// TIA Portal V17 export
// export: Created 2025-05-08T13:18:02.6118738Z, ExportSetting WithDefaults, DisplayName Totally Integrated Automation Portal, DisplayVersion V17 Update 8, DisplayName TIA Portal Openness, DisplayVersion V17 Update 8, DisplayName TIA Portal Version Control Interface, DisplayVersion V17, DisplayName SINAMICS Startdrive Advanced, DisplayVersion V17 SP2, DisplayName SINAMICS Startdrive G110M, G120, G120C, G120D, G120P, G115D, DisplayVersion V17 SP2, DisplayName SINAMICS Startdrive G130, G150, S120, S150, SINAMICS MV, S210, DisplayVersion V17 SP2, DisplayName STEP 7 Professional, DisplayVersion V17 Update 8, DisplayName SINUMERIK ONE STEP 7 Toolbox, DisplayVersion V17 Update 12, DisplayName SINUMERIK 840D sl STEP 7 Toolbox, DisplayVersion V17 Update 12, DisplayName STEP 7 Safety, DisplayVersion V17 Update 6, DisplayName WinCC Advanced, DisplayVersion V17 Update 8
FUNCTION "FC16016_METHOD_CALLS_U3_MEAS_STA_MEAS_R" : Void   // FC16016, LAD
{ S7_Optimized_Access := 'TRUE' }
VERSION : 0.1
// stored: AutoNumber false, IsIECCheckEnabled false, SetENOAutomatically false, UDAEnableTagReadback false
   VAR_TEMP
      AUX_WSTRING_PART_ID_MEAS_STA : WString;
      AUX_WCHARS : Array[0..63] of WChar;
      index : Int;
      AUX_ALARMS : Bool;
   END_VAR
   VAR CONSTANT
      VERSIONS_MAJOR : UInt := 2;
      VERSIONS_MINOR : UInt;
      FC_NUMBER : DInt := 16016;
   END_VAR
   VAR_TEMP   // added for the SCL form of the ladder/FBD networks
      _w1 : Bool;
      _w2 : Bool;
   END_VAR
BEGIN

REGION Network 1 (SCL): TRANSFORM TO WCHARS
   FOR #index := 0 TO 63 DO
       #AUX_WCHARS[#index] := CHAR_TO_WCHAR("DB8000_PART_STATUS".UNIT_3.FIXTURE_1.PART_A.PART_ID[#index]);
   END_FOR;
END_REGION

REGION Network 2: TRANSFORM TO WSTRING
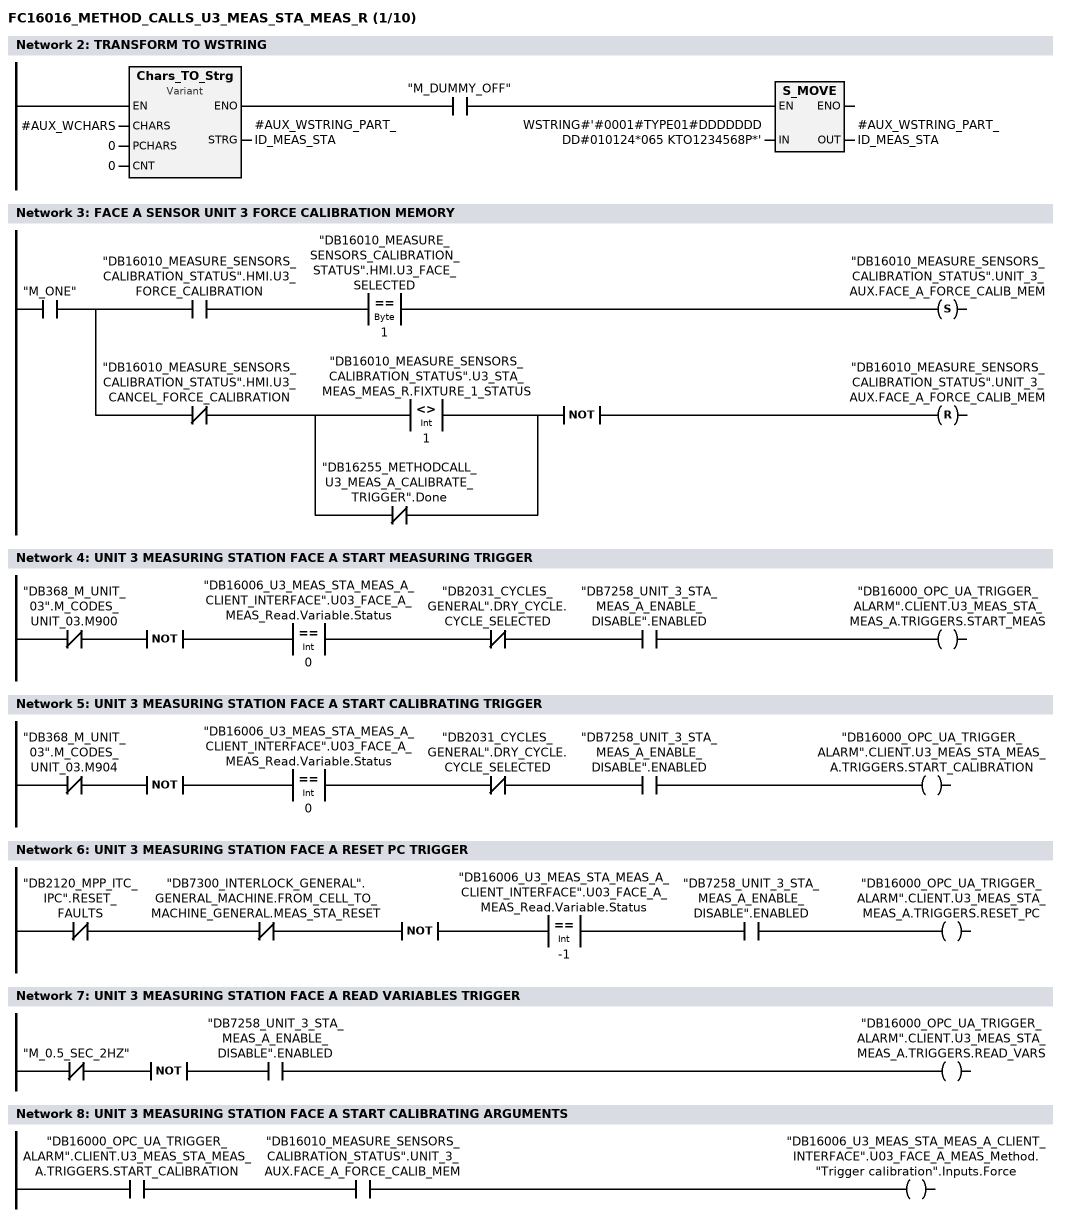
   RUNG wire#powerrail
      { S7_Templates := "[ptr_type := Variant, str_type := WString]" } Chars_TO_Strg(Chars := #AUX_WCHARS, pChars := 0, Cnt := 0, Strg => #AUX_WSTRING_PART_ID_MEAS_STA)
      Contact( "M_DUMMY_OFF" )
      S_Move(in := WSTRING#'#0001#TYPE01#DDDDDDDDD#010124*065 KTO1234568P*', out => #AUX_WSTRING_PART_ID_MEAS_STA)
   END_RUNG
   // the same network as SCL:
   Chars_TO_Strg(Chars := #AUX_WCHARS,
                 pChars := 0,
                 Cnt := 0,
                 Strg => #AUX_WSTRING_PART_ID_MEAS_STA,
                 ENO => #_w1);
   IF #_w1 AND "M_DUMMY_OFF" THEN
       #AUX_WSTRING_PART_ID_MEAS_STA := WSTRING#'#0001#TYPE01#DDDDDDDDD#010124*065 KTO1234568P*';
   END_IF;
END_REGION

REGION Network 3: FACE A SENSOR UNIT 3 FORCE CALIBRATION MEMORY
   RUNG wire#powerrail
      Contact( "M_ONE" )
      wire#w1
      Contact( "DB16010_MEASURE_SENSORS_CALIBRATION_STATUS".HMI.U3_FORCE_CALIBRATION )
      { S7_Templates := "SrcType := Byte" } EQ_Contact(in1 := "DB16010_MEASURE_SENSORS_CALIBRATION_STATUS".HMI.U3_FACE_SELECTED, in2 := 1)
      S_Coil( "DB16010_MEASURE_SENSORS_CALIBRATION_STATUS".UNIT_3_AUX.FACE_A_FORCE_CALIB_MEM )
   END_RUNG
   RUNG wire#w1
      I_Contact( "DB16010_MEASURE_SENSORS_CALIBRATION_STATUS".HMI.U3_CANCEL_FORCE_CALIBRATION )
      wire#w2
      { S7_Templates := "SrcType := Int" } NE_Contact(in1 := "DB16010_MEASURE_SENSORS_CALIBRATION_STATUS".U3_STA_MEAS_MEAS_R.FIXTURE_1_STATUS, in2 := 1)
      wire#w3
      Not()
      R_Coil( "DB16010_MEASURE_SENSORS_CALIBRATION_STATUS".UNIT_3_AUX.FACE_A_FORCE_CALIB_MEM )
   END_RUNG
   RUNG wire#w2
      I_Contact( "DB16255_METHODCALL_U3_MEAS_A_CALIBRATE_TRIGGER".Done )
   END_RUNG wire#w3
   // the same network as SCL:
   IF "M_ONE" AND "DB16010_MEASURE_SENSORS_CALIBRATION_STATUS".HMI.U3_FORCE_CALIBRATION AND ("DB16010_MEASURE_SENSORS_CALIBRATION_STATUS".HMI.U3_FACE_SELECTED = 1) THEN
       "DB16010_MEASURE_SENSORS_CALIBRATION_STATUS".UNIT_3_AUX.FACE_A_FORCE_CALIB_MEM := TRUE;
   END_IF;
   IF NOT ("M_ONE" AND NOT "DB16010_MEASURE_SENSORS_CALIBRATION_STATUS".HMI.U3_CANCEL_FORCE_CALIBRATION AND (("DB16010_MEASURE_SENSORS_CALIBRATION_STATUS".U3_STA_MEAS_MEAS_R.FIXTURE_1_STATUS <> 1) OR NOT "DB16255_METHODCALL_U3_MEAS_A_CALIBRATE_TRIGGER".Done)) THEN
       "DB16010_MEASURE_SENSORS_CALIBRATION_STATUS".UNIT_3_AUX.FACE_A_FORCE_CALIB_MEM := FALSE;
   END_IF;
END_REGION

REGION Network 4: UNIT 3 MEASURING STATION FACE A START MEASURING TRIGGER
   RUNG wire#powerrail
      I_Contact( "DB368_M_UNIT_03".M_CODES_UNIT_03.M900 )
      Not()
      { S7_Templates := "SrcType := Int" } EQ_Contact(in1 := "DB16006_U3_MEAS_STA_MEAS_A_CLIENT_INTERFACE".U03_FACE_A_MEAS_Read.Variable.Status, in2 := 0)
      I_Contact( "DB2031_CYCLES_GENERAL".DRY_CYCLE.CYCLE_SELECTED )
      Contact( "DB7258_UNIT_3_STA_MEAS_A_ENABLE_DISABLE".ENABLED )
      Coil( "DB16000_OPC_UA_TRIGGER_ALARM".CLIENT.U3_MEAS_STA_MEAS_A.TRIGGERS.START_MEAS )
   END_RUNG
   // the same network as SCL:
   "DB16000_OPC_UA_TRIGGER_ALARM".CLIENT.U3_MEAS_STA_MEAS_A.TRIGGERS.START_MEAS := NOT (NOT "DB368_M_UNIT_03".M_CODES_UNIT_03.M900) AND ("DB16006_U3_MEAS_STA_MEAS_A_CLIENT_INTERFACE".U03_FACE_A_MEAS_Read.Variable.Status = 0) AND NOT "DB2031_CYCLES_GENERAL".DRY_CYCLE.CYCLE_SELECTED AND "DB7258_UNIT_3_STA_MEAS_A_ENABLE_DISABLE".ENABLED;
END_REGION

REGION Network 5: UNIT 3 MEASURING STATION FACE A START CALIBRATING TRIGGER
   RUNG wire#powerrail
      I_Contact( "DB368_M_UNIT_03".M_CODES_UNIT_03.M904 )
      Not()
      { S7_Templates := "SrcType := Int" } EQ_Contact(in1 := "DB16006_U3_MEAS_STA_MEAS_A_CLIENT_INTERFACE".U03_FACE_A_MEAS_Read.Variable.Status, in2 := 0)
      I_Contact( "DB2031_CYCLES_GENERAL".DRY_CYCLE.CYCLE_SELECTED )
      Contact( "DB7258_UNIT_3_STA_MEAS_A_ENABLE_DISABLE".ENABLED )
      Coil( "DB16000_OPC_UA_TRIGGER_ALARM".CLIENT.U3_MEAS_STA_MEAS_A.TRIGGERS.START_CALIBRATION )
   END_RUNG
   // the same network as SCL:
   "DB16000_OPC_UA_TRIGGER_ALARM".CLIENT.U3_MEAS_STA_MEAS_A.TRIGGERS.START_CALIBRATION := NOT (NOT "DB368_M_UNIT_03".M_CODES_UNIT_03.M904) AND ("DB16006_U3_MEAS_STA_MEAS_A_CLIENT_INTERFACE".U03_FACE_A_MEAS_Read.Variable.Status = 0) AND NOT "DB2031_CYCLES_GENERAL".DRY_CYCLE.CYCLE_SELECTED AND "DB7258_UNIT_3_STA_MEAS_A_ENABLE_DISABLE".ENABLED;
END_REGION

REGION Network 6: UNIT 3 MEASURING STATION FACE A RESET PC TRIGGER
   RUNG wire#powerrail
      I_Contact( "DB2120_MPP_ITC_IPC".RESET_FAULTS )
      I_Contact( "DB7300_INTERLOCK_GENERAL".GENERAL_MACHINE.FROM_CELL_TO_MACHINE_GENERAL.MEAS_STA_RESET )
      Not()
      { S7_Templates := "SrcType := Int" } EQ_Contact(in1 := "DB16006_U3_MEAS_STA_MEAS_A_CLIENT_INTERFACE".U03_FACE_A_MEAS_Read.Variable.Status, in2 := -1)
      Contact( "DB7258_UNIT_3_STA_MEAS_A_ENABLE_DISABLE".ENABLED )
      Coil( "DB16000_OPC_UA_TRIGGER_ALARM".CLIENT.U3_MEAS_STA_MEAS_A.TRIGGERS.RESET_PC )
   END_RUNG
   // the same network as SCL:
   "DB16000_OPC_UA_TRIGGER_ALARM".CLIENT.U3_MEAS_STA_MEAS_A.TRIGGERS.RESET_PC := NOT (NOT "DB2120_MPP_ITC_IPC".RESET_FAULTS AND NOT "DB7300_INTERLOCK_GENERAL".GENERAL_MACHINE.FROM_CELL_TO_MACHINE_GENERAL.MEAS_STA_RESET) AND ("DB16006_U3_MEAS_STA_MEAS_A_CLIENT_INTERFACE".U03_FACE_A_MEAS_Read.Variable.Status = (-1)) AND "DB7258_UNIT_3_STA_MEAS_A_ENABLE_DISABLE".ENABLED;
END_REGION

REGION Network 7: UNIT 3 MEASURING STATION FACE A READ VARIABLES TRIGGER
   RUNG wire#powerrail
      I_Contact( "M_0.5_SEC_2HZ" )
      Not()
      Contact( "DB7258_UNIT_3_STA_MEAS_A_ENABLE_DISABLE".ENABLED )
      Coil( "DB16000_OPC_UA_TRIGGER_ALARM".CLIENT.U3_MEAS_STA_MEAS_A.TRIGGERS.READ_VARS )
   END_RUNG
   // the same network as SCL:
   "DB16000_OPC_UA_TRIGGER_ALARM".CLIENT.U3_MEAS_STA_MEAS_A.TRIGGERS.READ_VARS := NOT (NOT "M_0.5_SEC_2HZ") AND "DB7258_UNIT_3_STA_MEAS_A_ENABLE_DISABLE".ENABLED;
END_REGION

REGION Network 8: UNIT 3 MEASURING STATION FACE A START CALIBRATING ARGUMENTS
   RUNG wire#powerrail
      Contact( "DB16000_OPC_UA_TRIGGER_ALARM".CLIENT.U3_MEAS_STA_MEAS_A.TRIGGERS.START_CALIBRATION )
      Contact( "DB16010_MEASURE_SENSORS_CALIBRATION_STATUS".UNIT_3_AUX.FACE_A_FORCE_CALIB_MEM )
      Coil( "DB16006_U3_MEAS_STA_MEAS_A_CLIENT_INTERFACE".U03_FACE_A_MEAS_Method."Trigger calibration".Inputs.Force )
   END_RUNG
   // the same network as SCL:
   "DB16006_U3_MEAS_STA_MEAS_A_CLIENT_INTERFACE".U03_FACE_A_MEAS_Method."Trigger calibration".Inputs.Force := "DB16000_OPC_UA_TRIGGER_ALARM".CLIENT.U3_MEAS_STA_MEAS_A.TRIGGERS.START_CALIBRATION AND "DB16010_MEASURE_SENSORS_CALIBRATION_STATUS".UNIT_3_AUX.FACE_A_FORCE_CALIB_MEM;
END_REGION

REGION Network 9: UNIT 3 MEASURING STATION FACE A MEASURING TRIGGER CALL
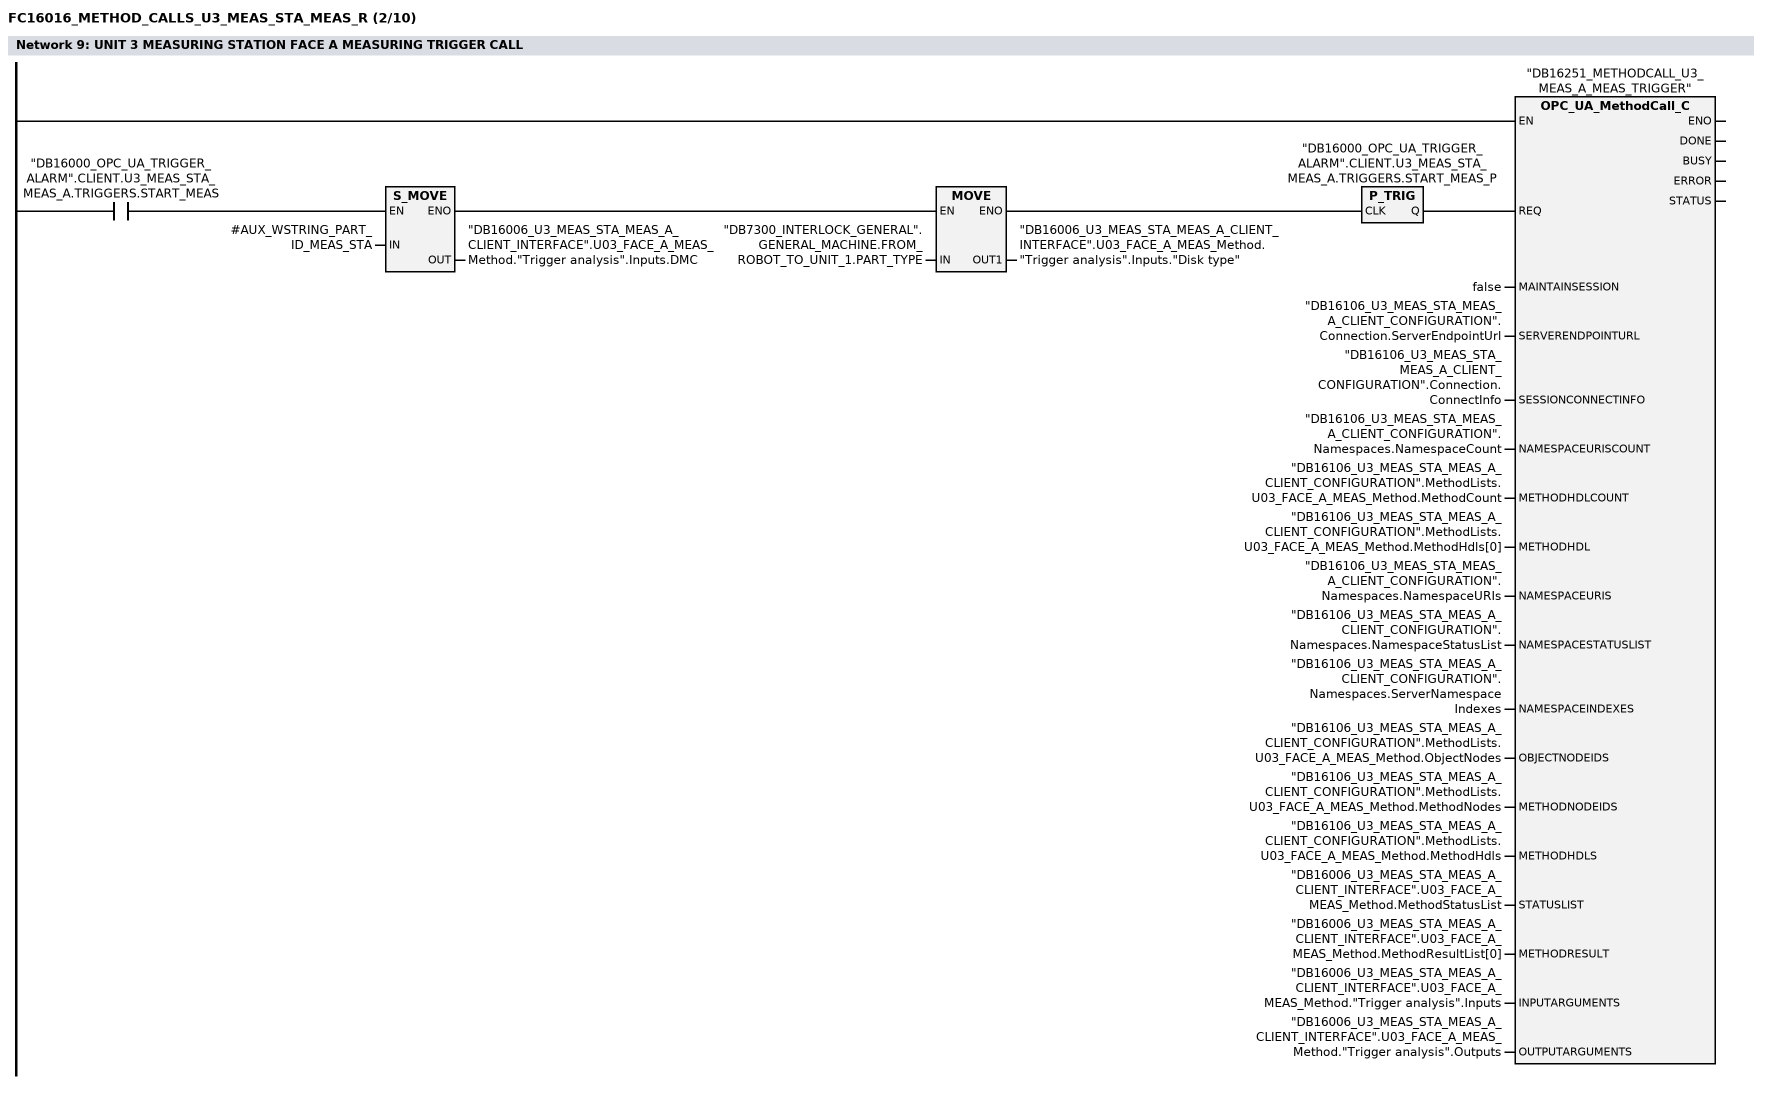
   RUNG wire#powerrail
      "DB16251_METHODCALL_U3_MEAS_A_MEAS_TRIGGER".OPC_UA_MethodCall_C(REQ := wire#w1, MaintainSession := false, ServerEndpointUrl := "DB16106_U3_MEAS_STA_MEAS_A_CLIENT_CONFIGURATION".Connection.ServerEndpointUrl, SessionConnectInfo := "DB16106_U3_MEAS_STA_MEAS_A_CLIENT_CONFIGURATION".Connection.ConnectInfo, NamespaceUrisCount := "DB16106_U3_MEAS_STA_MEAS_A_CLIENT_CONFIGURATION".Namespaces.NamespaceCount, MethodHdlCount := "DB16106_U3_MEAS_STA_MEAS_A_CLIENT_CONFIGURATION".MethodLists.U03_FACE_A_MEAS_Method.MethodCount, MethodHdl := "DB16106_U3_MEAS_STA_MEAS_A_CLIENT_CONFIGURATION".MethodLists.U03_FACE_A_MEAS_Method.MethodHdls[0], NamespaceUris := "DB16106_U3_MEAS_STA_MEAS_A_CLIENT_CONFIGURATION".Namespaces.NamespaceURIs, NamespaceStatusList := "DB16106_U3_MEAS_STA_MEAS_A_CLIENT_CONFIGURATION".Namespaces.NamespaceStatusList, NamespaceIndexes := "DB16106_U3_MEAS_STA_MEAS_A_CLIENT_CONFIGURATION".Namespaces.ServerNamespaceIndexes, ObjectNodeIDs := "DB16106_U3_MEAS_STA_MEAS_A_CLIENT_CONFIGURATION".MethodLists.U03_FACE_A_MEAS_Method.ObjectNodes, MethodNodeIDs := "DB16106_U3_MEAS_STA_MEAS_A_CLIENT_CONFIGURATION".MethodLists.U03_FACE_A_MEAS_Method.MethodNodes, MethodHdls := "DB16106_U3_MEAS_STA_MEAS_A_CLIENT_CONFIGURATION".MethodLists.U03_FACE_A_MEAS_Method.MethodHdls, StatusList := "DB16006_U3_MEAS_STA_MEAS_A_CLIENT_INTERFACE".U03_FACE_A_MEAS_Method.MethodStatusList, MethodResult := "DB16006_U3_MEAS_STA_MEAS_A_CLIENT_INTERFACE".U03_FACE_A_MEAS_Method.MethodResultList[0], InputArguments := "DB16006_U3_MEAS_STA_MEAS_A_CLIENT_INTERFACE".U03_FACE_A_MEAS_Method."Trigger analysis".Inputs, OutputArguments := "DB16006_U3_MEAS_STA_MEAS_A_CLIENT_INTERFACE".U03_FACE_A_MEAS_Method."Trigger analysis".Outputs, Done =>, Busy =>, Error =>, Status =>)
   END_RUNG
   RUNG wire#powerrail
      Contact( "DB16000_OPC_UA_TRIGGER_ALARM".CLIENT.U3_MEAS_STA_MEAS_A.TRIGGERS.START_MEAS )
      S_Move(in := #AUX_WSTRING_PART_ID_MEAS_STA, out => "DB16006_U3_MEAS_STA_MEAS_A_CLIENT_INTERFACE".U03_FACE_A_MEAS_Method."Trigger analysis".Inputs.DMC)
      Move(in := "DB7300_INTERLOCK_GENERAL".GENERAL_MACHINE.FROM_ROBOT_TO_UNIT_1.PART_TYPE, out1 => "DB16006_U3_MEAS_STA_MEAS_A_CLIENT_INTERFACE".U03_FACE_A_MEAS_Method."Trigger analysis".Inputs."Disk type")
      P_Trig( "DB16000_OPC_UA_TRIGGER_ALARM".CLIENT.U3_MEAS_STA_MEAS_A.TRIGGERS.START_MEAS_P )
   END_RUNG wire#w1
   // the same network as SCL:
   IF "DB16000_OPC_UA_TRIGGER_ALARM".CLIENT.U3_MEAS_STA_MEAS_A.TRIGGERS.START_MEAS THEN
       "DB16006_U3_MEAS_STA_MEAS_A_CLIENT_INTERFACE".U03_FACE_A_MEAS_Method."Trigger analysis".Inputs.DMC := #AUX_WSTRING_PART_ID_MEAS_STA;
       "DB16006_U3_MEAS_STA_MEAS_A_CLIENT_INTERFACE".U03_FACE_A_MEAS_Method."Trigger analysis".Inputs."Disk type" := "DB7300_INTERLOCK_GENERAL".GENERAL_MACHINE.FROM_ROBOT_TO_UNIT_1.PART_TYPE;
   END_IF;
   #_w1 := "DB16000_OPC_UA_TRIGGER_ALARM".CLIENT.U3_MEAS_STA_MEAS_A.TRIGGERS.START_MEAS AND NOT "DB16000_OPC_UA_TRIGGER_ALARM".CLIENT.U3_MEAS_STA_MEAS_A.TRIGGERS.START_MEAS_P;   // rising edge
   "DB16000_OPC_UA_TRIGGER_ALARM".CLIENT.U3_MEAS_STA_MEAS_A.TRIGGERS.START_MEAS_P := "DB16000_OPC_UA_TRIGGER_ALARM".CLIENT.U3_MEAS_STA_MEAS_A.TRIGGERS.START_MEAS;
   "DB16251_METHODCALL_U3_MEAS_A_MEAS_TRIGGER"(REQ := #_w1,   // OPC_UA_MethodCall_C
                           MaintainSession := false,
                           ServerEndpointUrl := "DB16106_U3_MEAS_STA_MEAS_A_CLIENT_CONFIGURATION".Connection.ServerEndpointUrl,
                           SessionConnectInfo := "DB16106_U3_MEAS_STA_MEAS_A_CLIENT_CONFIGURATION".Connection.ConnectInfo,
                           NamespaceUrisCount := "DB16106_U3_MEAS_STA_MEAS_A_CLIENT_CONFIGURATION".Namespaces.NamespaceCount,
                           MethodHdlCount := "DB16106_U3_MEAS_STA_MEAS_A_CLIENT_CONFIGURATION".MethodLists.U03_FACE_A_MEAS_Method.MethodCount,
                           MethodHdl := "DB16106_U3_MEAS_STA_MEAS_A_CLIENT_CONFIGURATION".MethodLists.U03_FACE_A_MEAS_Method.MethodHdls[0],
                           NamespaceUris := "DB16106_U3_MEAS_STA_MEAS_A_CLIENT_CONFIGURATION".Namespaces.NamespaceURIs,
                           NamespaceStatusList := "DB16106_U3_MEAS_STA_MEAS_A_CLIENT_CONFIGURATION".Namespaces.NamespaceStatusList,
                           NamespaceIndexes := "DB16106_U3_MEAS_STA_MEAS_A_CLIENT_CONFIGURATION".Namespaces.ServerNamespaceIndexes,
                           ObjectNodeIDs := "DB16106_U3_MEAS_STA_MEAS_A_CLIENT_CONFIGURATION".MethodLists.U03_FACE_A_MEAS_Method.ObjectNodes,
                           MethodNodeIDs := "DB16106_U3_MEAS_STA_MEAS_A_CLIENT_CONFIGURATION".MethodLists.U03_FACE_A_MEAS_Method.MethodNodes,
                           MethodHdls := "DB16106_U3_MEAS_STA_MEAS_A_CLIENT_CONFIGURATION".MethodLists.U03_FACE_A_MEAS_Method.MethodHdls,
                           StatusList := "DB16006_U3_MEAS_STA_MEAS_A_CLIENT_INTERFACE".U03_FACE_A_MEAS_Method.MethodStatusList,
                           MethodResult := "DB16006_U3_MEAS_STA_MEAS_A_CLIENT_INTERFACE".U03_FACE_A_MEAS_Method.MethodResultList[0],
                           InputArguments := "DB16006_U3_MEAS_STA_MEAS_A_CLIENT_INTERFACE".U03_FACE_A_MEAS_Method."Trigger analysis".Inputs,
                           OutputArguments := "DB16006_U3_MEAS_STA_MEAS_A_CLIENT_INTERFACE".U03_FACE_A_MEAS_Method."Trigger analysis".Outputs);
END_REGION

REGION Network 10: UNIT 3 MEASURING STATION FACE A CALIBRATING TRIGGER CALL
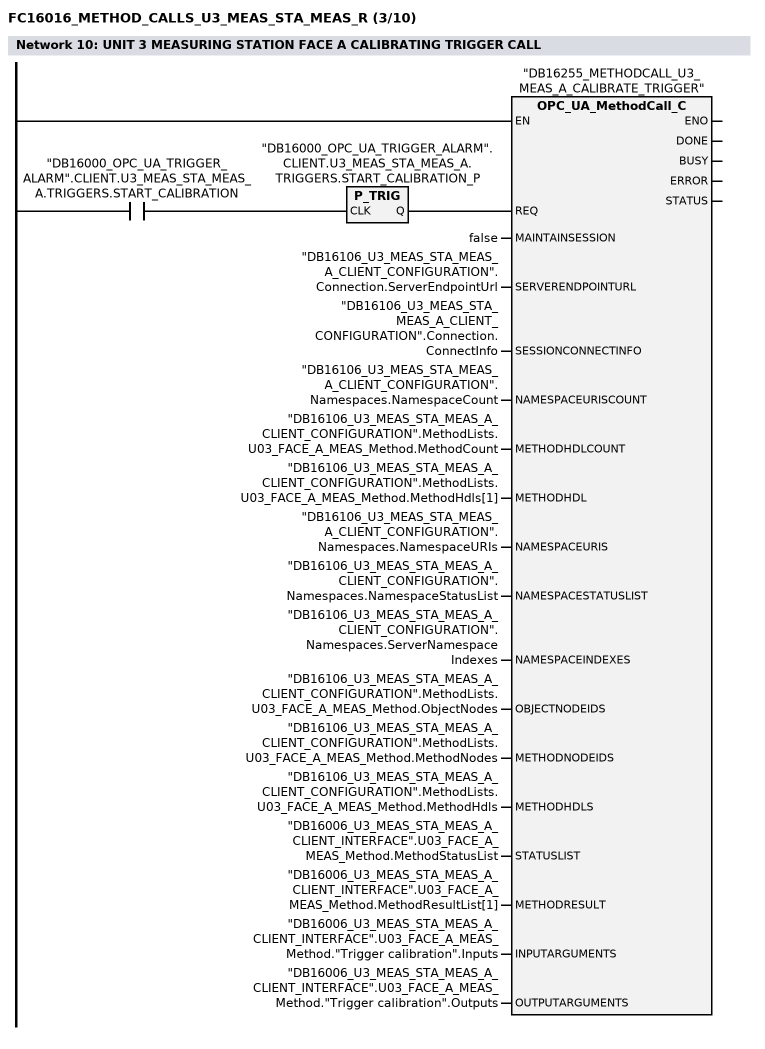
   RUNG wire#powerrail
      "DB16255_METHODCALL_U3_MEAS_A_CALIBRATE_TRIGGER".OPC_UA_MethodCall_C(REQ := wire#w1, MaintainSession := false, ServerEndpointUrl := "DB16106_U3_MEAS_STA_MEAS_A_CLIENT_CONFIGURATION".Connection.ServerEndpointUrl, SessionConnectInfo := "DB16106_U3_MEAS_STA_MEAS_A_CLIENT_CONFIGURATION".Connection.ConnectInfo, NamespaceUrisCount := "DB16106_U3_MEAS_STA_MEAS_A_CLIENT_CONFIGURATION".Namespaces.NamespaceCount, MethodHdlCount := "DB16106_U3_MEAS_STA_MEAS_A_CLIENT_CONFIGURATION".MethodLists.U03_FACE_A_MEAS_Method.MethodCount, MethodHdl := "DB16106_U3_MEAS_STA_MEAS_A_CLIENT_CONFIGURATION".MethodLists.U03_FACE_A_MEAS_Method.MethodHdls[1], NamespaceUris := "DB16106_U3_MEAS_STA_MEAS_A_CLIENT_CONFIGURATION".Namespaces.NamespaceURIs, NamespaceStatusList := "DB16106_U3_MEAS_STA_MEAS_A_CLIENT_CONFIGURATION".Namespaces.NamespaceStatusList, NamespaceIndexes := "DB16106_U3_MEAS_STA_MEAS_A_CLIENT_CONFIGURATION".Namespaces.ServerNamespaceIndexes, ObjectNodeIDs := "DB16106_U3_MEAS_STA_MEAS_A_CLIENT_CONFIGURATION".MethodLists.U03_FACE_A_MEAS_Method.ObjectNodes, MethodNodeIDs := "DB16106_U3_MEAS_STA_MEAS_A_CLIENT_CONFIGURATION".MethodLists.U03_FACE_A_MEAS_Method.MethodNodes, MethodHdls := "DB16106_U3_MEAS_STA_MEAS_A_CLIENT_CONFIGURATION".MethodLists.U03_FACE_A_MEAS_Method.MethodHdls, StatusList := "DB16006_U3_MEAS_STA_MEAS_A_CLIENT_INTERFACE".U03_FACE_A_MEAS_Method.MethodStatusList, MethodResult := "DB16006_U3_MEAS_STA_MEAS_A_CLIENT_INTERFACE".U03_FACE_A_MEAS_Method.MethodResultList[1], InputArguments := "DB16006_U3_MEAS_STA_MEAS_A_CLIENT_INTERFACE".U03_FACE_A_MEAS_Method."Trigger calibration".Inputs, OutputArguments := "DB16006_U3_MEAS_STA_MEAS_A_CLIENT_INTERFACE".U03_FACE_A_MEAS_Method."Trigger calibration".Outputs, Done =>, Busy =>, Error =>, Status =>)
   END_RUNG
   RUNG wire#powerrail
      Contact( "DB16000_OPC_UA_TRIGGER_ALARM".CLIENT.U3_MEAS_STA_MEAS_A.TRIGGERS.START_CALIBRATION )
      P_Trig( "DB16000_OPC_UA_TRIGGER_ALARM".CLIENT.U3_MEAS_STA_MEAS_A.TRIGGERS.START_CALIBRATION_P )
   END_RUNG wire#w1
   // the same network as SCL:
   #_w1 := "DB16000_OPC_UA_TRIGGER_ALARM".CLIENT.U3_MEAS_STA_MEAS_A.TRIGGERS.START_CALIBRATION AND NOT "DB16000_OPC_UA_TRIGGER_ALARM".CLIENT.U3_MEAS_STA_MEAS_A.TRIGGERS.START_CALIBRATION_P;   // rising edge
   "DB16000_OPC_UA_TRIGGER_ALARM".CLIENT.U3_MEAS_STA_MEAS_A.TRIGGERS.START_CALIBRATION_P := "DB16000_OPC_UA_TRIGGER_ALARM".CLIENT.U3_MEAS_STA_MEAS_A.TRIGGERS.START_CALIBRATION;
   "DB16255_METHODCALL_U3_MEAS_A_CALIBRATE_TRIGGER"(REQ := #_w1,   // OPC_UA_MethodCall_C
                           MaintainSession := false,
                           ServerEndpointUrl := "DB16106_U3_MEAS_STA_MEAS_A_CLIENT_CONFIGURATION".Connection.ServerEndpointUrl,
                           SessionConnectInfo := "DB16106_U3_MEAS_STA_MEAS_A_CLIENT_CONFIGURATION".Connection.ConnectInfo,
                           NamespaceUrisCount := "DB16106_U3_MEAS_STA_MEAS_A_CLIENT_CONFIGURATION".Namespaces.NamespaceCount,
                           MethodHdlCount := "DB16106_U3_MEAS_STA_MEAS_A_CLIENT_CONFIGURATION".MethodLists.U03_FACE_A_MEAS_Method.MethodCount,
                           MethodHdl := "DB16106_U3_MEAS_STA_MEAS_A_CLIENT_CONFIGURATION".MethodLists.U03_FACE_A_MEAS_Method.MethodHdls[1],
                           NamespaceUris := "DB16106_U3_MEAS_STA_MEAS_A_CLIENT_CONFIGURATION".Namespaces.NamespaceURIs,
                           NamespaceStatusList := "DB16106_U3_MEAS_STA_MEAS_A_CLIENT_CONFIGURATION".Namespaces.NamespaceStatusList,
                           NamespaceIndexes := "DB16106_U3_MEAS_STA_MEAS_A_CLIENT_CONFIGURATION".Namespaces.ServerNamespaceIndexes,
                           ObjectNodeIDs := "DB16106_U3_MEAS_STA_MEAS_A_CLIENT_CONFIGURATION".MethodLists.U03_FACE_A_MEAS_Method.ObjectNodes,
                           MethodNodeIDs := "DB16106_U3_MEAS_STA_MEAS_A_CLIENT_CONFIGURATION".MethodLists.U03_FACE_A_MEAS_Method.MethodNodes,
                           MethodHdls := "DB16106_U3_MEAS_STA_MEAS_A_CLIENT_CONFIGURATION".MethodLists.U03_FACE_A_MEAS_Method.MethodHdls,
                           StatusList := "DB16006_U3_MEAS_STA_MEAS_A_CLIENT_INTERFACE".U03_FACE_A_MEAS_Method.MethodStatusList,
                           MethodResult := "DB16006_U3_MEAS_STA_MEAS_A_CLIENT_INTERFACE".U03_FACE_A_MEAS_Method.MethodResultList[1],
                           InputArguments := "DB16006_U3_MEAS_STA_MEAS_A_CLIENT_INTERFACE".U03_FACE_A_MEAS_Method."Trigger calibration".Inputs,
                           OutputArguments := "DB16006_U3_MEAS_STA_MEAS_A_CLIENT_INTERFACE".U03_FACE_A_MEAS_Method."Trigger calibration".Outputs);
END_REGION

REGION Network 11: UNIT 3 MEASURING STATION FACE A RESET PC TRIGGER CALL
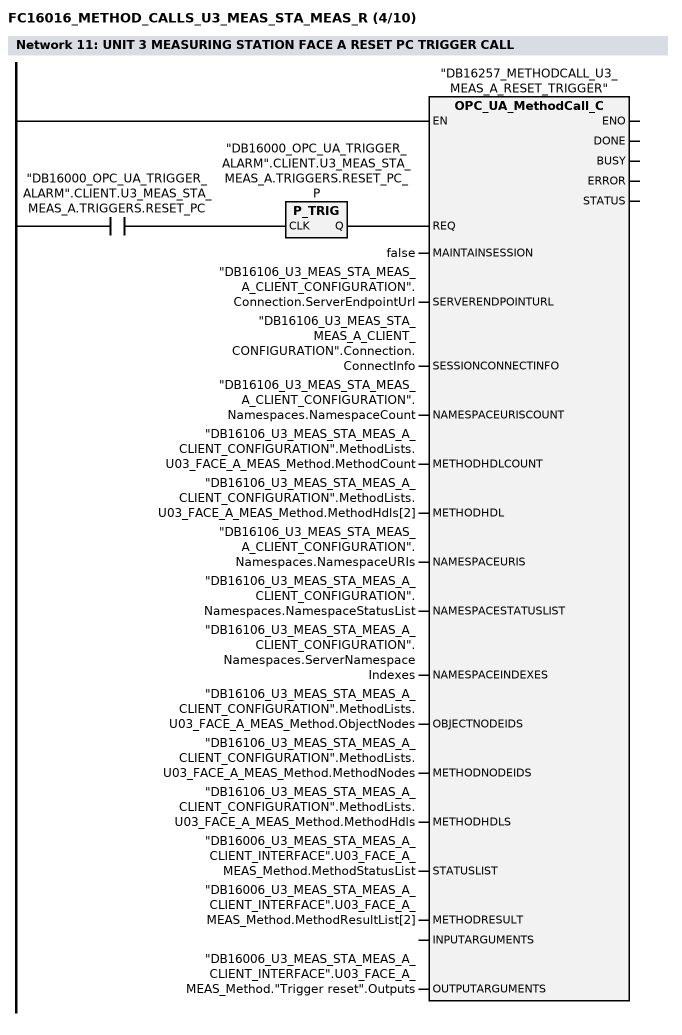
   RUNG wire#powerrail
      "DB16257_METHODCALL_U3_MEAS_A_RESET_TRIGGER".OPC_UA_MethodCall_C(REQ := wire#w1, MaintainSession := false, ServerEndpointUrl := "DB16106_U3_MEAS_STA_MEAS_A_CLIENT_CONFIGURATION".Connection.ServerEndpointUrl, SessionConnectInfo := "DB16106_U3_MEAS_STA_MEAS_A_CLIENT_CONFIGURATION".Connection.ConnectInfo, NamespaceUrisCount := "DB16106_U3_MEAS_STA_MEAS_A_CLIENT_CONFIGURATION".Namespaces.NamespaceCount, MethodHdlCount := "DB16106_U3_MEAS_STA_MEAS_A_CLIENT_CONFIGURATION".MethodLists.U03_FACE_A_MEAS_Method.MethodCount, MethodHdl := "DB16106_U3_MEAS_STA_MEAS_A_CLIENT_CONFIGURATION".MethodLists.U03_FACE_A_MEAS_Method.MethodHdls[2], NamespaceUris := "DB16106_U3_MEAS_STA_MEAS_A_CLIENT_CONFIGURATION".Namespaces.NamespaceURIs, NamespaceStatusList := "DB16106_U3_MEAS_STA_MEAS_A_CLIENT_CONFIGURATION".Namespaces.NamespaceStatusList, NamespaceIndexes := "DB16106_U3_MEAS_STA_MEAS_A_CLIENT_CONFIGURATION".Namespaces.ServerNamespaceIndexes, ObjectNodeIDs := "DB16106_U3_MEAS_STA_MEAS_A_CLIENT_CONFIGURATION".MethodLists.U03_FACE_A_MEAS_Method.ObjectNodes, MethodNodeIDs := "DB16106_U3_MEAS_STA_MEAS_A_CLIENT_CONFIGURATION".MethodLists.U03_FACE_A_MEAS_Method.MethodNodes, MethodHdls := "DB16106_U3_MEAS_STA_MEAS_A_CLIENT_CONFIGURATION".MethodLists.U03_FACE_A_MEAS_Method.MethodHdls, StatusList := "DB16006_U3_MEAS_STA_MEAS_A_CLIENT_INTERFACE".U03_FACE_A_MEAS_Method.MethodStatusList, MethodResult := "DB16006_U3_MEAS_STA_MEAS_A_CLIENT_INTERFACE".U03_FACE_A_MEAS_Method.MethodResultList[2], InputArguments :=, OutputArguments := "DB16006_U3_MEAS_STA_MEAS_A_CLIENT_INTERFACE".U03_FACE_A_MEAS_Method."Trigger reset".Outputs, Done =>, Busy =>, Error =>, Status =>)
   END_RUNG
   RUNG wire#powerrail
      Contact( "DB16000_OPC_UA_TRIGGER_ALARM".CLIENT.U3_MEAS_STA_MEAS_A.TRIGGERS.RESET_PC )
      P_Trig( "DB16000_OPC_UA_TRIGGER_ALARM".CLIENT.U3_MEAS_STA_MEAS_A.TRIGGERS.RESET_PC_P )
   END_RUNG wire#w1
   // the same network as SCL:
   #_w1 := "DB16000_OPC_UA_TRIGGER_ALARM".CLIENT.U3_MEAS_STA_MEAS_A.TRIGGERS.RESET_PC AND NOT "DB16000_OPC_UA_TRIGGER_ALARM".CLIENT.U3_MEAS_STA_MEAS_A.TRIGGERS.RESET_PC_P;   // rising edge
   "DB16000_OPC_UA_TRIGGER_ALARM".CLIENT.U3_MEAS_STA_MEAS_A.TRIGGERS.RESET_PC_P := "DB16000_OPC_UA_TRIGGER_ALARM".CLIENT.U3_MEAS_STA_MEAS_A.TRIGGERS.RESET_PC;
   "DB16257_METHODCALL_U3_MEAS_A_RESET_TRIGGER"(REQ := #_w1,   // OPC_UA_MethodCall_C
                           MaintainSession := false,
                           ServerEndpointUrl := "DB16106_U3_MEAS_STA_MEAS_A_CLIENT_CONFIGURATION".Connection.ServerEndpointUrl,
                           SessionConnectInfo := "DB16106_U3_MEAS_STA_MEAS_A_CLIENT_CONFIGURATION".Connection.ConnectInfo,
                           NamespaceUrisCount := "DB16106_U3_MEAS_STA_MEAS_A_CLIENT_CONFIGURATION".Namespaces.NamespaceCount,
                           MethodHdlCount := "DB16106_U3_MEAS_STA_MEAS_A_CLIENT_CONFIGURATION".MethodLists.U03_FACE_A_MEAS_Method.MethodCount,
                           MethodHdl := "DB16106_U3_MEAS_STA_MEAS_A_CLIENT_CONFIGURATION".MethodLists.U03_FACE_A_MEAS_Method.MethodHdls[2],
                           NamespaceUris := "DB16106_U3_MEAS_STA_MEAS_A_CLIENT_CONFIGURATION".Namespaces.NamespaceURIs,
                           NamespaceStatusList := "DB16106_U3_MEAS_STA_MEAS_A_CLIENT_CONFIGURATION".Namespaces.NamespaceStatusList,
                           NamespaceIndexes := "DB16106_U3_MEAS_STA_MEAS_A_CLIENT_CONFIGURATION".Namespaces.ServerNamespaceIndexes,
                           ObjectNodeIDs := "DB16106_U3_MEAS_STA_MEAS_A_CLIENT_CONFIGURATION".MethodLists.U03_FACE_A_MEAS_Method.ObjectNodes,
                           MethodNodeIDs := "DB16106_U3_MEAS_STA_MEAS_A_CLIENT_CONFIGURATION".MethodLists.U03_FACE_A_MEAS_Method.MethodNodes,
                           MethodHdls := "DB16106_U3_MEAS_STA_MEAS_A_CLIENT_CONFIGURATION".MethodLists.U03_FACE_A_MEAS_Method.MethodHdls,
                           StatusList := "DB16006_U3_MEAS_STA_MEAS_A_CLIENT_INTERFACE".U03_FACE_A_MEAS_Method.MethodStatusList,
                           MethodResult := "DB16006_U3_MEAS_STA_MEAS_A_CLIENT_INTERFACE".U03_FACE_A_MEAS_Method.MethodResultList[2],
                           OutputArguments := "DB16006_U3_MEAS_STA_MEAS_A_CLIENT_INTERFACE".U03_FACE_A_MEAS_Method."Trigger reset".Outputs);
END_REGION

REGION Network 12: UNIT 3 MEASURING STATION FACE A READ VARIABLES TRIGGER CALL
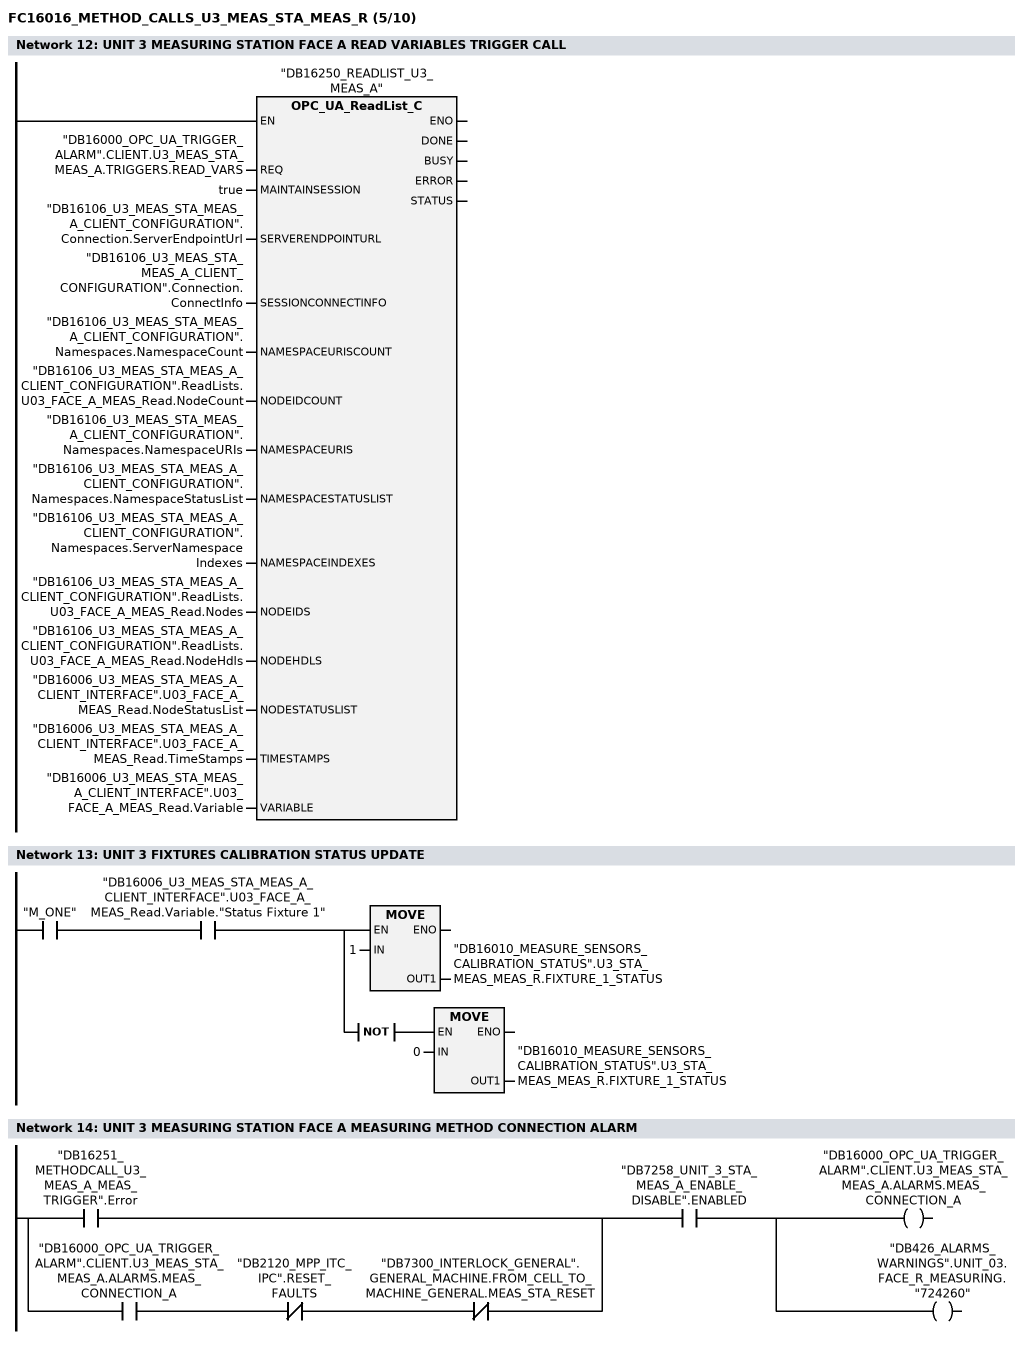
   RUNG wire#powerrail
      "DB16250_READLIST_U3_MEAS_A".OPC_UA_ReadList_C(REQ := "DB16000_OPC_UA_TRIGGER_ALARM".CLIENT.U3_MEAS_STA_MEAS_A.TRIGGERS.READ_VARS, MaintainSession := true, ServerEndpointUrl := "DB16106_U3_MEAS_STA_MEAS_A_CLIENT_CONFIGURATION".Connection.ServerEndpointUrl, SessionConnectInfo := "DB16106_U3_MEAS_STA_MEAS_A_CLIENT_CONFIGURATION".Connection.ConnectInfo, NamespaceUrisCount := "DB16106_U3_MEAS_STA_MEAS_A_CLIENT_CONFIGURATION".Namespaces.NamespaceCount, NodeIDCount := "DB16106_U3_MEAS_STA_MEAS_A_CLIENT_CONFIGURATION".ReadLists.U03_FACE_A_MEAS_Read.NodeCount, NamespaceUris := "DB16106_U3_MEAS_STA_MEAS_A_CLIENT_CONFIGURATION".Namespaces.NamespaceURIs, NamespaceStatusList := "DB16106_U3_MEAS_STA_MEAS_A_CLIENT_CONFIGURATION".Namespaces.NamespaceStatusList, NamespaceIndexes := "DB16106_U3_MEAS_STA_MEAS_A_CLIENT_CONFIGURATION".Namespaces.ServerNamespaceIndexes, NodeIDs := "DB16106_U3_MEAS_STA_MEAS_A_CLIENT_CONFIGURATION".ReadLists.U03_FACE_A_MEAS_Read.Nodes, NodeHdls := "DB16106_U3_MEAS_STA_MEAS_A_CLIENT_CONFIGURATION".ReadLists.U03_FACE_A_MEAS_Read.NodeHdls, NodeStatusList := "DB16006_U3_MEAS_STA_MEAS_A_CLIENT_INTERFACE".U03_FACE_A_MEAS_Read.NodeStatusList, Timestamps := "DB16006_U3_MEAS_STA_MEAS_A_CLIENT_INTERFACE".U03_FACE_A_MEAS_Read.TimeStamps, Variable := "DB16006_U3_MEAS_STA_MEAS_A_CLIENT_INTERFACE".U03_FACE_A_MEAS_Read.Variable, Done =>, Busy =>, Error =>, Status =>)
   END_RUNG
   // the same network as SCL:
   "DB16250_READLIST_U3_MEAS_A"(REQ := "DB16000_OPC_UA_TRIGGER_ALARM".CLIENT.U3_MEAS_STA_MEAS_A.TRIGGERS.READ_VARS,   // OPC_UA_ReadList_C
                           MaintainSession := true,
                           ServerEndpointUrl := "DB16106_U3_MEAS_STA_MEAS_A_CLIENT_CONFIGURATION".Connection.ServerEndpointUrl,
                           SessionConnectInfo := "DB16106_U3_MEAS_STA_MEAS_A_CLIENT_CONFIGURATION".Connection.ConnectInfo,
                           NamespaceUrisCount := "DB16106_U3_MEAS_STA_MEAS_A_CLIENT_CONFIGURATION".Namespaces.NamespaceCount,
                           NodeIDCount := "DB16106_U3_MEAS_STA_MEAS_A_CLIENT_CONFIGURATION".ReadLists.U03_FACE_A_MEAS_Read.NodeCount,
                           NamespaceUris := "DB16106_U3_MEAS_STA_MEAS_A_CLIENT_CONFIGURATION".Namespaces.NamespaceURIs,
                           NamespaceStatusList := "DB16106_U3_MEAS_STA_MEAS_A_CLIENT_CONFIGURATION".Namespaces.NamespaceStatusList,
                           NamespaceIndexes := "DB16106_U3_MEAS_STA_MEAS_A_CLIENT_CONFIGURATION".Namespaces.ServerNamespaceIndexes,
                           NodeIDs := "DB16106_U3_MEAS_STA_MEAS_A_CLIENT_CONFIGURATION".ReadLists.U03_FACE_A_MEAS_Read.Nodes,
                           NodeHdls := "DB16106_U3_MEAS_STA_MEAS_A_CLIENT_CONFIGURATION".ReadLists.U03_FACE_A_MEAS_Read.NodeHdls,
                           NodeStatusList := "DB16006_U3_MEAS_STA_MEAS_A_CLIENT_INTERFACE".U03_FACE_A_MEAS_Read.NodeStatusList,
                           Timestamps := "DB16006_U3_MEAS_STA_MEAS_A_CLIENT_INTERFACE".U03_FACE_A_MEAS_Read.TimeStamps,
                           Variable := "DB16006_U3_MEAS_STA_MEAS_A_CLIENT_INTERFACE".U03_FACE_A_MEAS_Read.Variable);
END_REGION

REGION Network 13: UNIT 3 FIXTURES CALIBRATION STATUS UPDATE
   RUNG wire#powerrail
      Contact( "M_ONE" )
      Contact( "DB16006_U3_MEAS_STA_MEAS_A_CLIENT_INTERFACE".U03_FACE_A_MEAS_Read.Variable."Status Fixture 1" )
      wire#w1
      Move(in := 1, out1 => "DB16010_MEASURE_SENSORS_CALIBRATION_STATUS".U3_STA_MEAS_MEAS_R.FIXTURE_1_STATUS)
   END_RUNG
   RUNG wire#w1
      Not()
      Move(in := 0, out1 => "DB16010_MEASURE_SENSORS_CALIBRATION_STATUS".U3_STA_MEAS_MEAS_R.FIXTURE_1_STATUS)
   END_RUNG
   // the same network as SCL:
   #_w1 := "M_ONE" AND "DB16006_U3_MEAS_STA_MEAS_A_CLIENT_INTERFACE".U03_FACE_A_MEAS_Read.Variable."Status Fixture 1";
   IF #_w1 THEN
       "DB16010_MEASURE_SENSORS_CALIBRATION_STATUS".U3_STA_MEAS_MEAS_R.FIXTURE_1_STATUS := 1;
   END_IF;
   IF NOT #_w1 THEN
       "DB16010_MEASURE_SENSORS_CALIBRATION_STATUS".U3_STA_MEAS_MEAS_R.FIXTURE_1_STATUS := 0;
   END_IF;
END_REGION

REGION Network 14: UNIT 3 MEASURING STATION FACE A MEASURING METHOD CONNECTION ALARM
   RUNG wire#powerrail
      Contact( "DB16251_METHODCALL_U3_MEAS_A_MEAS_TRIGGER".Error )
      wire#w1
      Contact( "DB7258_UNIT_3_STA_MEAS_A_ENABLE_DISABLE".ENABLED )
      wire#w2
      Coil( "DB16000_OPC_UA_TRIGGER_ALARM".CLIENT.U3_MEAS_STA_MEAS_A.ALARMS.MEAS_CONNECTION_A )
   END_RUNG
   RUNG wire#powerrail
      Contact( "DB16000_OPC_UA_TRIGGER_ALARM".CLIENT.U3_MEAS_STA_MEAS_A.ALARMS.MEAS_CONNECTION_A )
      I_Contact( "DB2120_MPP_ITC_IPC".RESET_FAULTS )
      I_Contact( "DB7300_INTERLOCK_GENERAL".GENERAL_MACHINE.FROM_CELL_TO_MACHINE_GENERAL.MEAS_STA_RESET )
   END_RUNG wire#w1
   RUNG wire#w2
      Coil( "DB426_ALARMS_WARNINGS".UNIT_03.FACE_R_MEASURING."724260" )
   END_RUNG
   // the same network as SCL:
   "DB16000_OPC_UA_TRIGGER_ALARM".CLIENT.U3_MEAS_STA_MEAS_A.ALARMS.MEAS_CONNECTION_A := ("DB16251_METHODCALL_U3_MEAS_A_MEAS_TRIGGER".Error OR ("DB16000_OPC_UA_TRIGGER_ALARM".CLIENT.U3_MEAS_STA_MEAS_A.ALARMS.MEAS_CONNECTION_A AND NOT "DB2120_MPP_ITC_IPC".RESET_FAULTS AND NOT "DB7300_INTERLOCK_GENERAL".GENERAL_MACHINE.FROM_CELL_TO_MACHINE_GENERAL.MEAS_STA_RESET)) AND "DB7258_UNIT_3_STA_MEAS_A_ENABLE_DISABLE".ENABLED;
   "DB426_ALARMS_WARNINGS".UNIT_03.FACE_R_MEASURING."724260" := "DB16000_OPC_UA_TRIGGER_ALARM".CLIENT.U3_MEAS_STA_MEAS_A.ALARMS.MEAS_CONNECTION_A;
END_REGION

REGION Network 15: UNIT 3 MEASURING STATION FACE A MEASURING METHOD WORKING OR BLOCKED ALARM
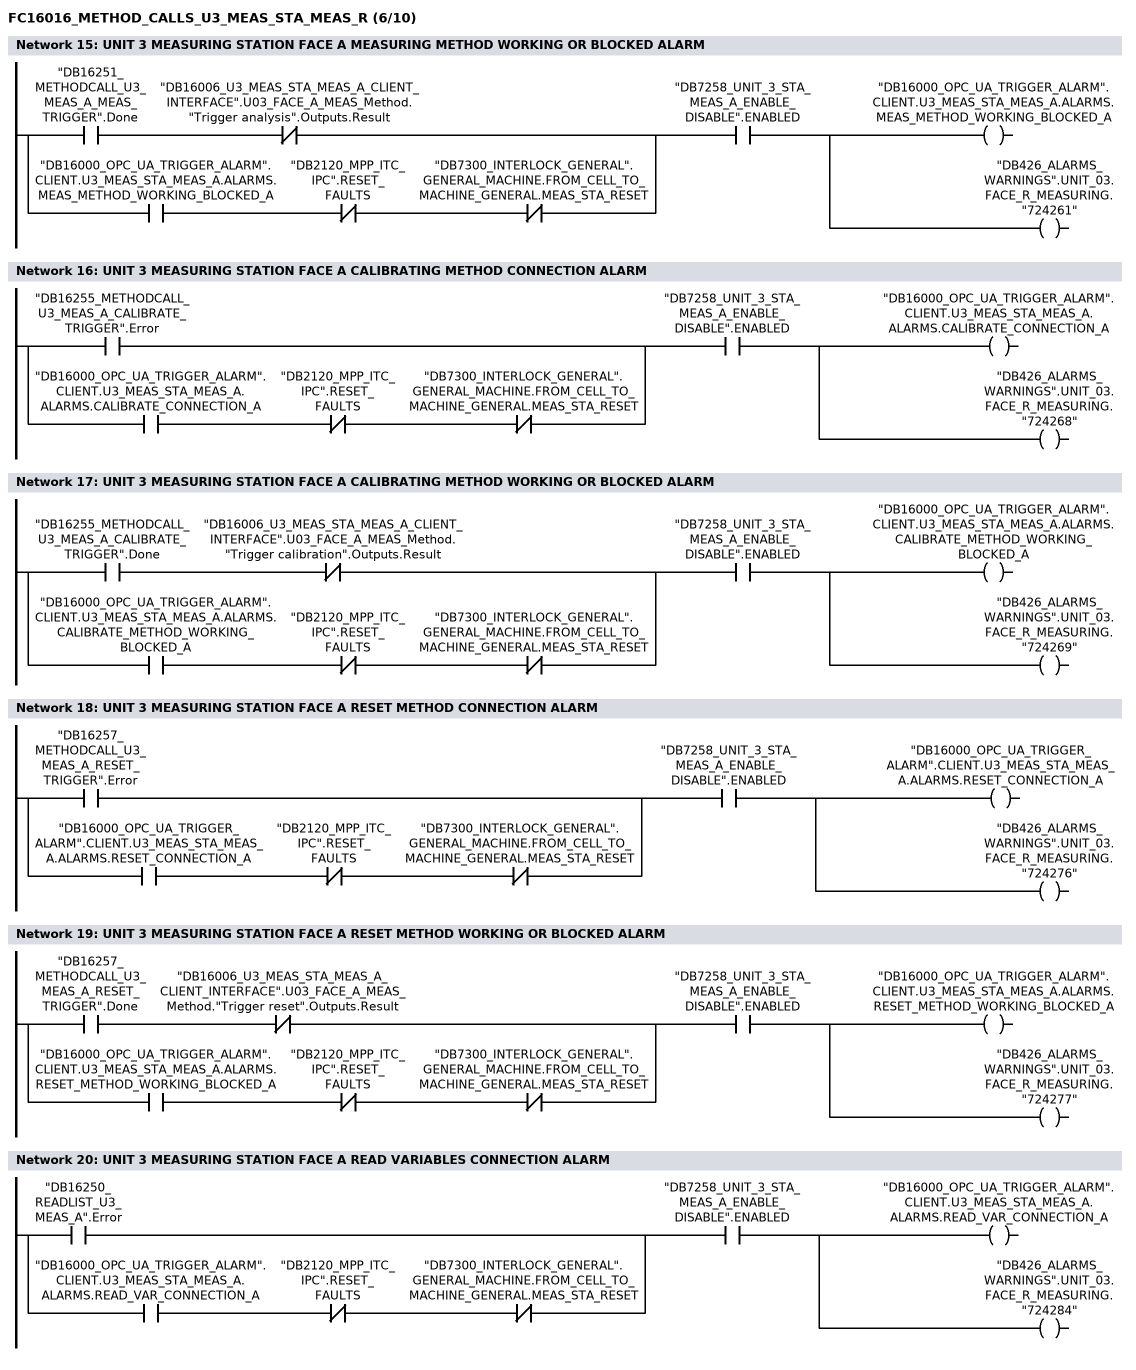
   RUNG wire#powerrail
      Contact( "DB16251_METHODCALL_U3_MEAS_A_MEAS_TRIGGER".Done )
      I_Contact( "DB16006_U3_MEAS_STA_MEAS_A_CLIENT_INTERFACE".U03_FACE_A_MEAS_Method."Trigger analysis".Outputs.Result )
      wire#w1
      Contact( "DB7258_UNIT_3_STA_MEAS_A_ENABLE_DISABLE".ENABLED )
      wire#w2
      Coil( "DB16000_OPC_UA_TRIGGER_ALARM".CLIENT.U3_MEAS_STA_MEAS_A.ALARMS.MEAS_METHOD_WORKING_BLOCKED_A )
   END_RUNG
   RUNG wire#powerrail
      Contact( "DB16000_OPC_UA_TRIGGER_ALARM".CLIENT.U3_MEAS_STA_MEAS_A.ALARMS.MEAS_METHOD_WORKING_BLOCKED_A )
      I_Contact( "DB2120_MPP_ITC_IPC".RESET_FAULTS )
      I_Contact( "DB7300_INTERLOCK_GENERAL".GENERAL_MACHINE.FROM_CELL_TO_MACHINE_GENERAL.MEAS_STA_RESET )
   END_RUNG wire#w1
   RUNG wire#w2
      Coil( "DB426_ALARMS_WARNINGS".UNIT_03.FACE_R_MEASURING."724261" )
   END_RUNG
   // the same network as SCL:
   "DB16000_OPC_UA_TRIGGER_ALARM".CLIENT.U3_MEAS_STA_MEAS_A.ALARMS.MEAS_METHOD_WORKING_BLOCKED_A := (("DB16251_METHODCALL_U3_MEAS_A_MEAS_TRIGGER".Done AND NOT "DB16006_U3_MEAS_STA_MEAS_A_CLIENT_INTERFACE".U03_FACE_A_MEAS_Method."Trigger analysis".Outputs.Result) OR ("DB16000_OPC_UA_TRIGGER_ALARM".CLIENT.U3_MEAS_STA_MEAS_A.ALARMS.MEAS_METHOD_WORKING_BLOCKED_A AND NOT "DB2120_MPP_ITC_IPC".RESET_FAULTS AND NOT "DB7300_INTERLOCK_GENERAL".GENERAL_MACHINE.FROM_CELL_TO_MACHINE_GENERAL.MEAS_STA_RESET)) AND "DB7258_UNIT_3_STA_MEAS_A_ENABLE_DISABLE".ENABLED;
   "DB426_ALARMS_WARNINGS".UNIT_03.FACE_R_MEASURING."724261" := "DB16000_OPC_UA_TRIGGER_ALARM".CLIENT.U3_MEAS_STA_MEAS_A.ALARMS.MEAS_METHOD_WORKING_BLOCKED_A;
END_REGION

REGION Network 16: UNIT 3 MEASURING STATION FACE A CALIBRATING METHOD CONNECTION ALARM
   RUNG wire#powerrail
      Contact( "DB16255_METHODCALL_U3_MEAS_A_CALIBRATE_TRIGGER".Error )
      wire#w1
      Contact( "DB7258_UNIT_3_STA_MEAS_A_ENABLE_DISABLE".ENABLED )
      wire#w2
      Coil( "DB16000_OPC_UA_TRIGGER_ALARM".CLIENT.U3_MEAS_STA_MEAS_A.ALARMS.CALIBRATE_CONNECTION_A )
   END_RUNG
   RUNG wire#powerrail
      Contact( "DB16000_OPC_UA_TRIGGER_ALARM".CLIENT.U3_MEAS_STA_MEAS_A.ALARMS.CALIBRATE_CONNECTION_A )
      I_Contact( "DB2120_MPP_ITC_IPC".RESET_FAULTS )
      I_Contact( "DB7300_INTERLOCK_GENERAL".GENERAL_MACHINE.FROM_CELL_TO_MACHINE_GENERAL.MEAS_STA_RESET )
   END_RUNG wire#w1
   RUNG wire#w2
      Coil( "DB426_ALARMS_WARNINGS".UNIT_03.FACE_R_MEASURING."724268" )
   END_RUNG
   // the same network as SCL:
   "DB16000_OPC_UA_TRIGGER_ALARM".CLIENT.U3_MEAS_STA_MEAS_A.ALARMS.CALIBRATE_CONNECTION_A := ("DB16255_METHODCALL_U3_MEAS_A_CALIBRATE_TRIGGER".Error OR ("DB16000_OPC_UA_TRIGGER_ALARM".CLIENT.U3_MEAS_STA_MEAS_A.ALARMS.CALIBRATE_CONNECTION_A AND NOT "DB2120_MPP_ITC_IPC".RESET_FAULTS AND NOT "DB7300_INTERLOCK_GENERAL".GENERAL_MACHINE.FROM_CELL_TO_MACHINE_GENERAL.MEAS_STA_RESET)) AND "DB7258_UNIT_3_STA_MEAS_A_ENABLE_DISABLE".ENABLED;
   "DB426_ALARMS_WARNINGS".UNIT_03.FACE_R_MEASURING."724268" := "DB16000_OPC_UA_TRIGGER_ALARM".CLIENT.U3_MEAS_STA_MEAS_A.ALARMS.CALIBRATE_CONNECTION_A;
END_REGION

REGION Network 17: UNIT 3 MEASURING STATION FACE A CALIBRATING METHOD WORKING OR BLOCKED ALARM
   RUNG wire#powerrail
      Contact( "DB16255_METHODCALL_U3_MEAS_A_CALIBRATE_TRIGGER".Done )
      I_Contact( "DB16006_U3_MEAS_STA_MEAS_A_CLIENT_INTERFACE".U03_FACE_A_MEAS_Method."Trigger calibration".Outputs.Result )
      wire#w1
      Contact( "DB7258_UNIT_3_STA_MEAS_A_ENABLE_DISABLE".ENABLED )
      wire#w2
      Coil( "DB16000_OPC_UA_TRIGGER_ALARM".CLIENT.U3_MEAS_STA_MEAS_A.ALARMS.CALIBRATE_METHOD_WORKING_BLOCKED_A )
   END_RUNG
   RUNG wire#powerrail
      Contact( "DB16000_OPC_UA_TRIGGER_ALARM".CLIENT.U3_MEAS_STA_MEAS_A.ALARMS.CALIBRATE_METHOD_WORKING_BLOCKED_A )
      I_Contact( "DB2120_MPP_ITC_IPC".RESET_FAULTS )
      I_Contact( "DB7300_INTERLOCK_GENERAL".GENERAL_MACHINE.FROM_CELL_TO_MACHINE_GENERAL.MEAS_STA_RESET )
   END_RUNG wire#w1
   RUNG wire#w2
      Coil( "DB426_ALARMS_WARNINGS".UNIT_03.FACE_R_MEASURING."724269" )
   END_RUNG
   // the same network as SCL:
   "DB16000_OPC_UA_TRIGGER_ALARM".CLIENT.U3_MEAS_STA_MEAS_A.ALARMS.CALIBRATE_METHOD_WORKING_BLOCKED_A := (("DB16255_METHODCALL_U3_MEAS_A_CALIBRATE_TRIGGER".Done AND NOT "DB16006_U3_MEAS_STA_MEAS_A_CLIENT_INTERFACE".U03_FACE_A_MEAS_Method."Trigger calibration".Outputs.Result) OR ("DB16000_OPC_UA_TRIGGER_ALARM".CLIENT.U3_MEAS_STA_MEAS_A.ALARMS.CALIBRATE_METHOD_WORKING_BLOCKED_A AND NOT "DB2120_MPP_ITC_IPC".RESET_FAULTS AND NOT "DB7300_INTERLOCK_GENERAL".GENERAL_MACHINE.FROM_CELL_TO_MACHINE_GENERAL.MEAS_STA_RESET)) AND "DB7258_UNIT_3_STA_MEAS_A_ENABLE_DISABLE".ENABLED;
   "DB426_ALARMS_WARNINGS".UNIT_03.FACE_R_MEASURING."724269" := "DB16000_OPC_UA_TRIGGER_ALARM".CLIENT.U3_MEAS_STA_MEAS_A.ALARMS.CALIBRATE_METHOD_WORKING_BLOCKED_A;
END_REGION

REGION Network 18: UNIT 3 MEASURING STATION FACE A RESET METHOD CONNECTION ALARM
   RUNG wire#powerrail
      Contact( "DB16257_METHODCALL_U3_MEAS_A_RESET_TRIGGER".Error )
      wire#w1
      Contact( "DB7258_UNIT_3_STA_MEAS_A_ENABLE_DISABLE".ENABLED )
      wire#w2
      Coil( "DB16000_OPC_UA_TRIGGER_ALARM".CLIENT.U3_MEAS_STA_MEAS_A.ALARMS.RESET_CONNECTION_A )
   END_RUNG
   RUNG wire#powerrail
      Contact( "DB16000_OPC_UA_TRIGGER_ALARM".CLIENT.U3_MEAS_STA_MEAS_A.ALARMS.RESET_CONNECTION_A )
      I_Contact( "DB2120_MPP_ITC_IPC".RESET_FAULTS )
      I_Contact( "DB7300_INTERLOCK_GENERAL".GENERAL_MACHINE.FROM_CELL_TO_MACHINE_GENERAL.MEAS_STA_RESET )
   END_RUNG wire#w1
   RUNG wire#w2
      Coil( "DB426_ALARMS_WARNINGS".UNIT_03.FACE_R_MEASURING."724276" )
   END_RUNG
   // the same network as SCL:
   "DB16000_OPC_UA_TRIGGER_ALARM".CLIENT.U3_MEAS_STA_MEAS_A.ALARMS.RESET_CONNECTION_A := ("DB16257_METHODCALL_U3_MEAS_A_RESET_TRIGGER".Error OR ("DB16000_OPC_UA_TRIGGER_ALARM".CLIENT.U3_MEAS_STA_MEAS_A.ALARMS.RESET_CONNECTION_A AND NOT "DB2120_MPP_ITC_IPC".RESET_FAULTS AND NOT "DB7300_INTERLOCK_GENERAL".GENERAL_MACHINE.FROM_CELL_TO_MACHINE_GENERAL.MEAS_STA_RESET)) AND "DB7258_UNIT_3_STA_MEAS_A_ENABLE_DISABLE".ENABLED;
   "DB426_ALARMS_WARNINGS".UNIT_03.FACE_R_MEASURING."724276" := "DB16000_OPC_UA_TRIGGER_ALARM".CLIENT.U3_MEAS_STA_MEAS_A.ALARMS.RESET_CONNECTION_A;
END_REGION

REGION Network 19: UNIT 3 MEASURING STATION FACE A RESET METHOD WORKING OR BLOCKED ALARM
   RUNG wire#powerrail
      Contact( "DB16257_METHODCALL_U3_MEAS_A_RESET_TRIGGER".Done )
      I_Contact( "DB16006_U3_MEAS_STA_MEAS_A_CLIENT_INTERFACE".U03_FACE_A_MEAS_Method."Trigger reset".Outputs.Result )
      wire#w1
      Contact( "DB7258_UNIT_3_STA_MEAS_A_ENABLE_DISABLE".ENABLED )
      wire#w2
      Coil( "DB16000_OPC_UA_TRIGGER_ALARM".CLIENT.U3_MEAS_STA_MEAS_A.ALARMS.RESET_METHOD_WORKING_BLOCKED_A )
   END_RUNG
   RUNG wire#powerrail
      Contact( "DB16000_OPC_UA_TRIGGER_ALARM".CLIENT.U3_MEAS_STA_MEAS_A.ALARMS.RESET_METHOD_WORKING_BLOCKED_A )
      I_Contact( "DB2120_MPP_ITC_IPC".RESET_FAULTS )
      I_Contact( "DB7300_INTERLOCK_GENERAL".GENERAL_MACHINE.FROM_CELL_TO_MACHINE_GENERAL.MEAS_STA_RESET )
   END_RUNG wire#w1
   RUNG wire#w2
      Coil( "DB426_ALARMS_WARNINGS".UNIT_03.FACE_R_MEASURING."724277" )
   END_RUNG
   // the same network as SCL:
   "DB16000_OPC_UA_TRIGGER_ALARM".CLIENT.U3_MEAS_STA_MEAS_A.ALARMS.RESET_METHOD_WORKING_BLOCKED_A := (("DB16257_METHODCALL_U3_MEAS_A_RESET_TRIGGER".Done AND NOT "DB16006_U3_MEAS_STA_MEAS_A_CLIENT_INTERFACE".U03_FACE_A_MEAS_Method."Trigger reset".Outputs.Result) OR ("DB16000_OPC_UA_TRIGGER_ALARM".CLIENT.U3_MEAS_STA_MEAS_A.ALARMS.RESET_METHOD_WORKING_BLOCKED_A AND NOT "DB2120_MPP_ITC_IPC".RESET_FAULTS AND NOT "DB7300_INTERLOCK_GENERAL".GENERAL_MACHINE.FROM_CELL_TO_MACHINE_GENERAL.MEAS_STA_RESET)) AND "DB7258_UNIT_3_STA_MEAS_A_ENABLE_DISABLE".ENABLED;
   "DB426_ALARMS_WARNINGS".UNIT_03.FACE_R_MEASURING."724277" := "DB16000_OPC_UA_TRIGGER_ALARM".CLIENT.U3_MEAS_STA_MEAS_A.ALARMS.RESET_METHOD_WORKING_BLOCKED_A;
END_REGION

REGION Network 20: UNIT 3 MEASURING STATION FACE A READ VARIABLES CONNECTION ALARM
   RUNG wire#powerrail
      Contact( "DB16250_READLIST_U3_MEAS_A".Error )
      wire#w1
      Contact( "DB7258_UNIT_3_STA_MEAS_A_ENABLE_DISABLE".ENABLED )
      wire#w2
      Coil( "DB16000_OPC_UA_TRIGGER_ALARM".CLIENT.U3_MEAS_STA_MEAS_A.ALARMS.READ_VAR_CONNECTION_A )
   END_RUNG
   RUNG wire#powerrail
      Contact( "DB16000_OPC_UA_TRIGGER_ALARM".CLIENT.U3_MEAS_STA_MEAS_A.ALARMS.READ_VAR_CONNECTION_A )
      I_Contact( "DB2120_MPP_ITC_IPC".RESET_FAULTS )
      I_Contact( "DB7300_INTERLOCK_GENERAL".GENERAL_MACHINE.FROM_CELL_TO_MACHINE_GENERAL.MEAS_STA_RESET )
   END_RUNG wire#w1
   RUNG wire#w2
      Coil( "DB426_ALARMS_WARNINGS".UNIT_03.FACE_R_MEASURING."724284" )
   END_RUNG
   // the same network as SCL:
   "DB16000_OPC_UA_TRIGGER_ALARM".CLIENT.U3_MEAS_STA_MEAS_A.ALARMS.READ_VAR_CONNECTION_A := ("DB16250_READLIST_U3_MEAS_A".Error OR ("DB16000_OPC_UA_TRIGGER_ALARM".CLIENT.U3_MEAS_STA_MEAS_A.ALARMS.READ_VAR_CONNECTION_A AND NOT "DB2120_MPP_ITC_IPC".RESET_FAULTS AND NOT "DB7300_INTERLOCK_GENERAL".GENERAL_MACHINE.FROM_CELL_TO_MACHINE_GENERAL.MEAS_STA_RESET)) AND "DB7258_UNIT_3_STA_MEAS_A_ENABLE_DISABLE".ENABLED;
   "DB426_ALARMS_WARNINGS".UNIT_03.FACE_R_MEASURING."724284" := "DB16000_OPC_UA_TRIGGER_ALARM".CLIENT.U3_MEAS_STA_MEAS_A.ALARMS.READ_VAR_CONNECTION_A;
END_REGION

REGION Network 21: UNIT 3 MEASURING STATION FACE A READ VARIABLES WORKING OR BLOCKED ALARM
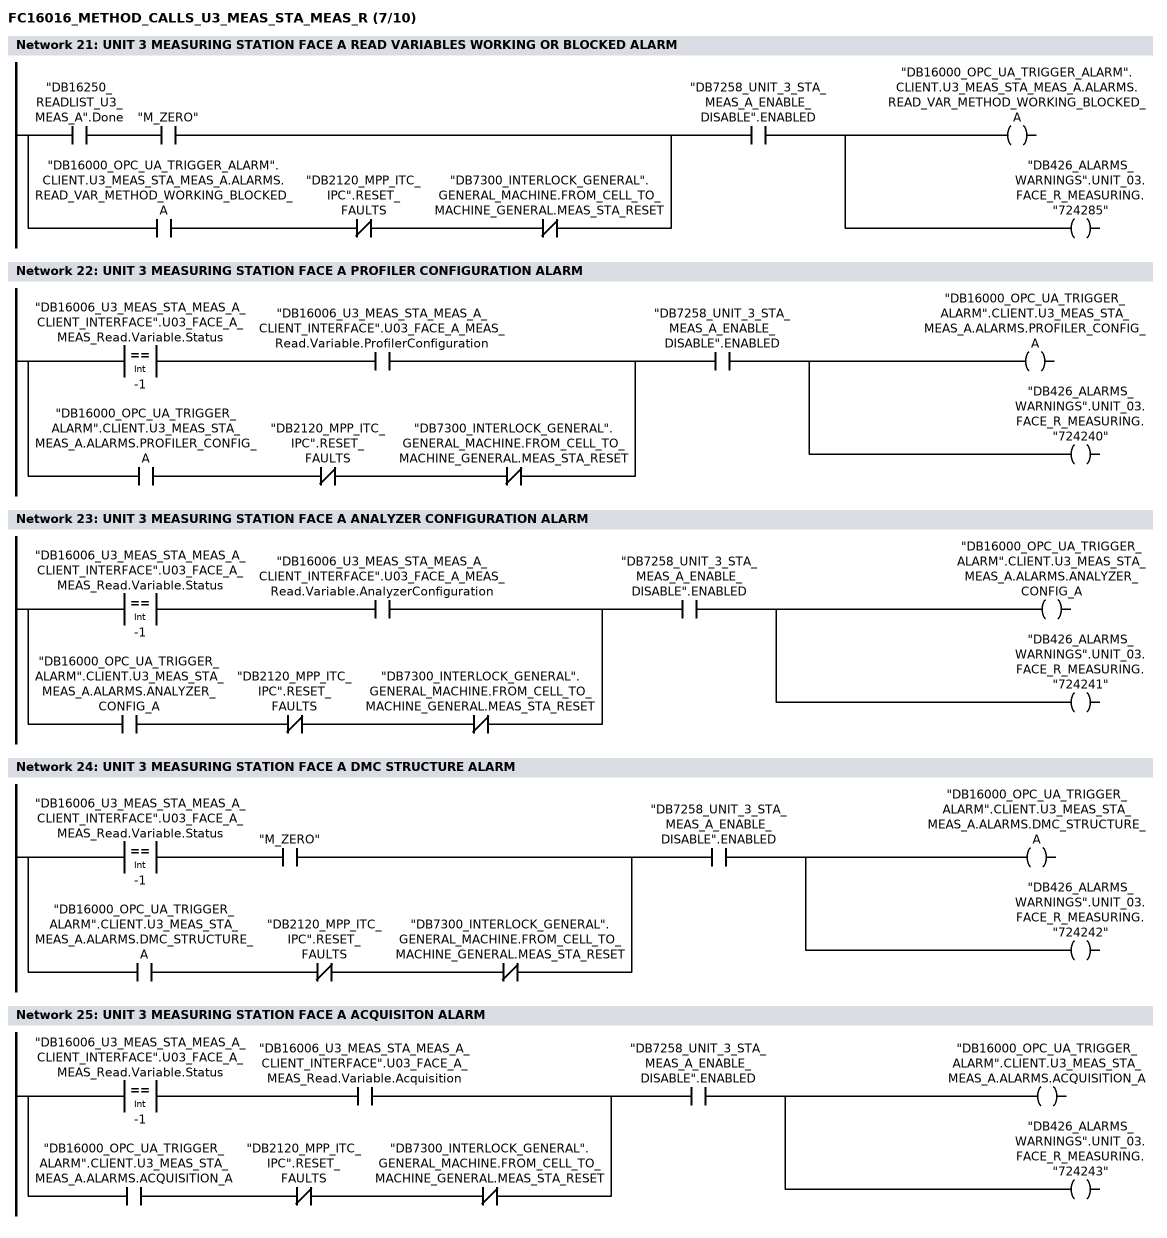
   RUNG wire#powerrail
      Contact( "DB16250_READLIST_U3_MEAS_A".Done )
      Contact( "M_ZERO" )
      wire#w1
      Contact( "DB7258_UNIT_3_STA_MEAS_A_ENABLE_DISABLE".ENABLED )
      wire#w2
      Coil( "DB16000_OPC_UA_TRIGGER_ALARM".CLIENT.U3_MEAS_STA_MEAS_A.ALARMS.READ_VAR_METHOD_WORKING_BLOCKED_A )
   END_RUNG
   RUNG wire#powerrail
      Contact( "DB16000_OPC_UA_TRIGGER_ALARM".CLIENT.U3_MEAS_STA_MEAS_A.ALARMS.READ_VAR_METHOD_WORKING_BLOCKED_A )
      I_Contact( "DB2120_MPP_ITC_IPC".RESET_FAULTS )
      I_Contact( "DB7300_INTERLOCK_GENERAL".GENERAL_MACHINE.FROM_CELL_TO_MACHINE_GENERAL.MEAS_STA_RESET )
   END_RUNG wire#w1
   RUNG wire#w2
      Coil( "DB426_ALARMS_WARNINGS".UNIT_03.FACE_R_MEASURING."724285" )
   END_RUNG
   // the same network as SCL:
   "DB16000_OPC_UA_TRIGGER_ALARM".CLIENT.U3_MEAS_STA_MEAS_A.ALARMS.READ_VAR_METHOD_WORKING_BLOCKED_A := (("DB16250_READLIST_U3_MEAS_A".Done AND "M_ZERO") OR ("DB16000_OPC_UA_TRIGGER_ALARM".CLIENT.U3_MEAS_STA_MEAS_A.ALARMS.READ_VAR_METHOD_WORKING_BLOCKED_A AND NOT "DB2120_MPP_ITC_IPC".RESET_FAULTS AND NOT "DB7300_INTERLOCK_GENERAL".GENERAL_MACHINE.FROM_CELL_TO_MACHINE_GENERAL.MEAS_STA_RESET)) AND "DB7258_UNIT_3_STA_MEAS_A_ENABLE_DISABLE".ENABLED;
   "DB426_ALARMS_WARNINGS".UNIT_03.FACE_R_MEASURING."724285" := "DB16000_OPC_UA_TRIGGER_ALARM".CLIENT.U3_MEAS_STA_MEAS_A.ALARMS.READ_VAR_METHOD_WORKING_BLOCKED_A;
END_REGION

REGION Network 22: UNIT 3 MEASURING STATION FACE A PROFILER CONFIGURATION ALARM
   RUNG wire#powerrail
      { S7_Templates := "SrcType := Int" } EQ_Contact(in1 := "DB16006_U3_MEAS_STA_MEAS_A_CLIENT_INTERFACE".U03_FACE_A_MEAS_Read.Variable.Status, in2 := -1)
      Contact( "DB16006_U3_MEAS_STA_MEAS_A_CLIENT_INTERFACE".U03_FACE_A_MEAS_Read.Variable.ProfilerConfiguration )
      wire#w1
      Contact( "DB7258_UNIT_3_STA_MEAS_A_ENABLE_DISABLE".ENABLED )
      wire#w2
      Coil( "DB16000_OPC_UA_TRIGGER_ALARM".CLIENT.U3_MEAS_STA_MEAS_A.ALARMS.PROFILER_CONFIG_A )
   END_RUNG
   RUNG wire#powerrail
      Contact( "DB16000_OPC_UA_TRIGGER_ALARM".CLIENT.U3_MEAS_STA_MEAS_A.ALARMS.PROFILER_CONFIG_A )
      I_Contact( "DB2120_MPP_ITC_IPC".RESET_FAULTS )
      I_Contact( "DB7300_INTERLOCK_GENERAL".GENERAL_MACHINE.FROM_CELL_TO_MACHINE_GENERAL.MEAS_STA_RESET )
   END_RUNG wire#w1
   RUNG wire#w2
      Coil( "DB426_ALARMS_WARNINGS".UNIT_03.FACE_R_MEASURING."724240" )
   END_RUNG
   // the same network as SCL:
   "DB16000_OPC_UA_TRIGGER_ALARM".CLIENT.U3_MEAS_STA_MEAS_A.ALARMS.PROFILER_CONFIG_A := ((("DB16006_U3_MEAS_STA_MEAS_A_CLIENT_INTERFACE".U03_FACE_A_MEAS_Read.Variable.Status = (-1)) AND "DB16006_U3_MEAS_STA_MEAS_A_CLIENT_INTERFACE".U03_FACE_A_MEAS_Read.Variable.ProfilerConfiguration) OR ("DB16000_OPC_UA_TRIGGER_ALARM".CLIENT.U3_MEAS_STA_MEAS_A.ALARMS.PROFILER_CONFIG_A AND NOT "DB2120_MPP_ITC_IPC".RESET_FAULTS AND NOT "DB7300_INTERLOCK_GENERAL".GENERAL_MACHINE.FROM_CELL_TO_MACHINE_GENERAL.MEAS_STA_RESET)) AND "DB7258_UNIT_3_STA_MEAS_A_ENABLE_DISABLE".ENABLED;
   "DB426_ALARMS_WARNINGS".UNIT_03.FACE_R_MEASURING."724240" := "DB16000_OPC_UA_TRIGGER_ALARM".CLIENT.U3_MEAS_STA_MEAS_A.ALARMS.PROFILER_CONFIG_A;
END_REGION

REGION Network 23: UNIT 3 MEASURING STATION FACE A ANALYZER CONFIGURATION ALARM
   RUNG wire#powerrail
      { S7_Templates := "SrcType := Int" } EQ_Contact(in1 := "DB16006_U3_MEAS_STA_MEAS_A_CLIENT_INTERFACE".U03_FACE_A_MEAS_Read.Variable.Status, in2 := -1)
      Contact( "DB16006_U3_MEAS_STA_MEAS_A_CLIENT_INTERFACE".U03_FACE_A_MEAS_Read.Variable.AnalyzerConfiguration )
      wire#w1
      Contact( "DB7258_UNIT_3_STA_MEAS_A_ENABLE_DISABLE".ENABLED )
      wire#w2
      Coil( "DB16000_OPC_UA_TRIGGER_ALARM".CLIENT.U3_MEAS_STA_MEAS_A.ALARMS.ANALYZER_CONFIG_A )
   END_RUNG
   RUNG wire#powerrail
      Contact( "DB16000_OPC_UA_TRIGGER_ALARM".CLIENT.U3_MEAS_STA_MEAS_A.ALARMS.ANALYZER_CONFIG_A )
      I_Contact( "DB2120_MPP_ITC_IPC".RESET_FAULTS )
      I_Contact( "DB7300_INTERLOCK_GENERAL".GENERAL_MACHINE.FROM_CELL_TO_MACHINE_GENERAL.MEAS_STA_RESET )
   END_RUNG wire#w1
   RUNG wire#w2
      Coil( "DB426_ALARMS_WARNINGS".UNIT_03.FACE_R_MEASURING."724241" )
   END_RUNG
   // the same network as SCL:
   "DB16000_OPC_UA_TRIGGER_ALARM".CLIENT.U3_MEAS_STA_MEAS_A.ALARMS.ANALYZER_CONFIG_A := ((("DB16006_U3_MEAS_STA_MEAS_A_CLIENT_INTERFACE".U03_FACE_A_MEAS_Read.Variable.Status = (-1)) AND "DB16006_U3_MEAS_STA_MEAS_A_CLIENT_INTERFACE".U03_FACE_A_MEAS_Read.Variable.AnalyzerConfiguration) OR ("DB16000_OPC_UA_TRIGGER_ALARM".CLIENT.U3_MEAS_STA_MEAS_A.ALARMS.ANALYZER_CONFIG_A AND NOT "DB2120_MPP_ITC_IPC".RESET_FAULTS AND NOT "DB7300_INTERLOCK_GENERAL".GENERAL_MACHINE.FROM_CELL_TO_MACHINE_GENERAL.MEAS_STA_RESET)) AND "DB7258_UNIT_3_STA_MEAS_A_ENABLE_DISABLE".ENABLED;
   "DB426_ALARMS_WARNINGS".UNIT_03.FACE_R_MEASURING."724241" := "DB16000_OPC_UA_TRIGGER_ALARM".CLIENT.U3_MEAS_STA_MEAS_A.ALARMS.ANALYZER_CONFIG_A;
END_REGION

REGION Network 24: UNIT 3 MEASURING STATION FACE A DMC STRUCTURE ALARM
   RUNG wire#powerrail
      { S7_Templates := "SrcType := Int" } EQ_Contact(in1 := "DB16006_U3_MEAS_STA_MEAS_A_CLIENT_INTERFACE".U03_FACE_A_MEAS_Read.Variable.Status, in2 := -1)
      Contact( "M_ZERO" )
      wire#w1
      Contact( "DB7258_UNIT_3_STA_MEAS_A_ENABLE_DISABLE".ENABLED )
      wire#w2
      Coil( "DB16000_OPC_UA_TRIGGER_ALARM".CLIENT.U3_MEAS_STA_MEAS_A.ALARMS.DMC_STRUCTURE_A )
   END_RUNG
   RUNG wire#powerrail
      Contact( "DB16000_OPC_UA_TRIGGER_ALARM".CLIENT.U3_MEAS_STA_MEAS_A.ALARMS.DMC_STRUCTURE_A )
      I_Contact( "DB2120_MPP_ITC_IPC".RESET_FAULTS )
      I_Contact( "DB7300_INTERLOCK_GENERAL".GENERAL_MACHINE.FROM_CELL_TO_MACHINE_GENERAL.MEAS_STA_RESET )
   END_RUNG wire#w1
   RUNG wire#w2
      Coil( "DB426_ALARMS_WARNINGS".UNIT_03.FACE_R_MEASURING."724242" )
   END_RUNG
   // the same network as SCL:
   "DB16000_OPC_UA_TRIGGER_ALARM".CLIENT.U3_MEAS_STA_MEAS_A.ALARMS.DMC_STRUCTURE_A := ((("DB16006_U3_MEAS_STA_MEAS_A_CLIENT_INTERFACE".U03_FACE_A_MEAS_Read.Variable.Status = (-1)) AND "M_ZERO") OR ("DB16000_OPC_UA_TRIGGER_ALARM".CLIENT.U3_MEAS_STA_MEAS_A.ALARMS.DMC_STRUCTURE_A AND NOT "DB2120_MPP_ITC_IPC".RESET_FAULTS AND NOT "DB7300_INTERLOCK_GENERAL".GENERAL_MACHINE.FROM_CELL_TO_MACHINE_GENERAL.MEAS_STA_RESET)) AND "DB7258_UNIT_3_STA_MEAS_A_ENABLE_DISABLE".ENABLED;
   "DB426_ALARMS_WARNINGS".UNIT_03.FACE_R_MEASURING."724242" := "DB16000_OPC_UA_TRIGGER_ALARM".CLIENT.U3_MEAS_STA_MEAS_A.ALARMS.DMC_STRUCTURE_A;
END_REGION

REGION Network 25: UNIT 3 MEASURING STATION FACE A ACQUISITON ALARM
   RUNG wire#powerrail
      { S7_Templates := "SrcType := Int" } EQ_Contact(in1 := "DB16006_U3_MEAS_STA_MEAS_A_CLIENT_INTERFACE".U03_FACE_A_MEAS_Read.Variable.Status, in2 := -1)
      Contact( "DB16006_U3_MEAS_STA_MEAS_A_CLIENT_INTERFACE".U03_FACE_A_MEAS_Read.Variable.Acquisition )
      wire#w1
      Contact( "DB7258_UNIT_3_STA_MEAS_A_ENABLE_DISABLE".ENABLED )
      wire#w2
      Coil( "DB16000_OPC_UA_TRIGGER_ALARM".CLIENT.U3_MEAS_STA_MEAS_A.ALARMS.ACQUISITION_A )
   END_RUNG
   RUNG wire#powerrail
      Contact( "DB16000_OPC_UA_TRIGGER_ALARM".CLIENT.U3_MEAS_STA_MEAS_A.ALARMS.ACQUISITION_A )
      I_Contact( "DB2120_MPP_ITC_IPC".RESET_FAULTS )
      I_Contact( "DB7300_INTERLOCK_GENERAL".GENERAL_MACHINE.FROM_CELL_TO_MACHINE_GENERAL.MEAS_STA_RESET )
   END_RUNG wire#w1
   RUNG wire#w2
      Coil( "DB426_ALARMS_WARNINGS".UNIT_03.FACE_R_MEASURING."724243" )
   END_RUNG
   // the same network as SCL:
   "DB16000_OPC_UA_TRIGGER_ALARM".CLIENT.U3_MEAS_STA_MEAS_A.ALARMS.ACQUISITION_A := ((("DB16006_U3_MEAS_STA_MEAS_A_CLIENT_INTERFACE".U03_FACE_A_MEAS_Read.Variable.Status = (-1)) AND "DB16006_U3_MEAS_STA_MEAS_A_CLIENT_INTERFACE".U03_FACE_A_MEAS_Read.Variable.Acquisition) OR ("DB16000_OPC_UA_TRIGGER_ALARM".CLIENT.U3_MEAS_STA_MEAS_A.ALARMS.ACQUISITION_A AND NOT "DB2120_MPP_ITC_IPC".RESET_FAULTS AND NOT "DB7300_INTERLOCK_GENERAL".GENERAL_MACHINE.FROM_CELL_TO_MACHINE_GENERAL.MEAS_STA_RESET)) AND "DB7258_UNIT_3_STA_MEAS_A_ENABLE_DISABLE".ENABLED;
   "DB426_ALARMS_WARNINGS".UNIT_03.FACE_R_MEASURING."724243" := "DB16000_OPC_UA_TRIGGER_ALARM".CLIENT.U3_MEAS_STA_MEAS_A.ALARMS.ACQUISITION_A;
END_REGION

REGION Network 26: UNIT 3 MEASURING STATION FACE A PROFILER INITIALIZTION ALARM
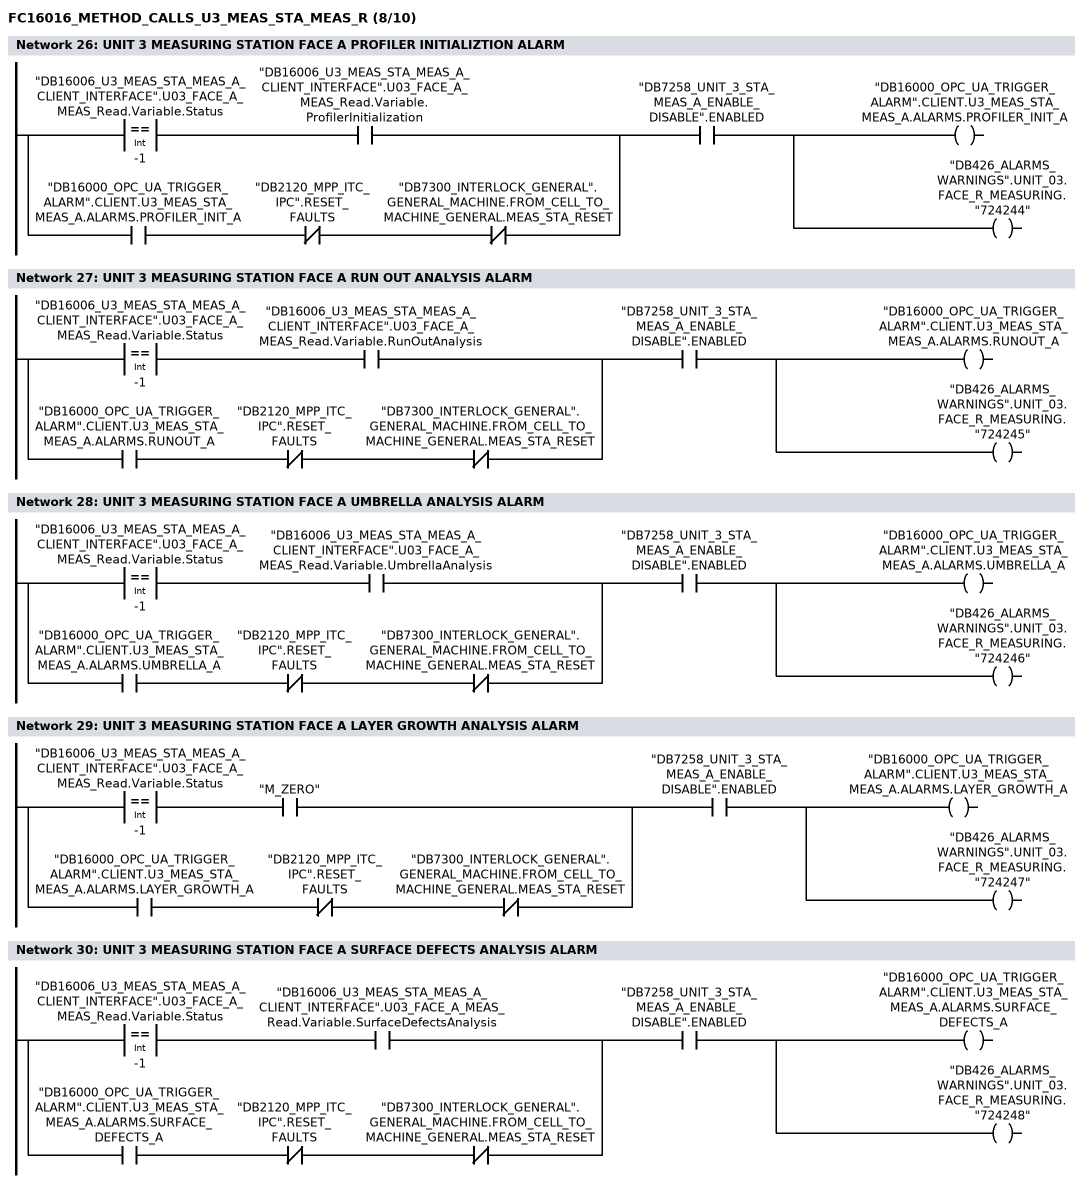
   RUNG wire#powerrail
      { S7_Templates := "SrcType := Int" } EQ_Contact(in1 := "DB16006_U3_MEAS_STA_MEAS_A_CLIENT_INTERFACE".U03_FACE_A_MEAS_Read.Variable.Status, in2 := -1)
      Contact( "DB16006_U3_MEAS_STA_MEAS_A_CLIENT_INTERFACE".U03_FACE_A_MEAS_Read.Variable.ProfilerInitialization )
      wire#w1
      Contact( "DB7258_UNIT_3_STA_MEAS_A_ENABLE_DISABLE".ENABLED )
      wire#w2
      Coil( "DB16000_OPC_UA_TRIGGER_ALARM".CLIENT.U3_MEAS_STA_MEAS_A.ALARMS.PROFILER_INIT_A )
   END_RUNG
   RUNG wire#powerrail
      Contact( "DB16000_OPC_UA_TRIGGER_ALARM".CLIENT.U3_MEAS_STA_MEAS_A.ALARMS.PROFILER_INIT_A )
      I_Contact( "DB2120_MPP_ITC_IPC".RESET_FAULTS )
      I_Contact( "DB7300_INTERLOCK_GENERAL".GENERAL_MACHINE.FROM_CELL_TO_MACHINE_GENERAL.MEAS_STA_RESET )
   END_RUNG wire#w1
   RUNG wire#w2
      Coil( "DB426_ALARMS_WARNINGS".UNIT_03.FACE_R_MEASURING."724244" )
   END_RUNG
   // the same network as SCL:
   "DB16000_OPC_UA_TRIGGER_ALARM".CLIENT.U3_MEAS_STA_MEAS_A.ALARMS.PROFILER_INIT_A := ((("DB16006_U3_MEAS_STA_MEAS_A_CLIENT_INTERFACE".U03_FACE_A_MEAS_Read.Variable.Status = (-1)) AND "DB16006_U3_MEAS_STA_MEAS_A_CLIENT_INTERFACE".U03_FACE_A_MEAS_Read.Variable.ProfilerInitialization) OR ("DB16000_OPC_UA_TRIGGER_ALARM".CLIENT.U3_MEAS_STA_MEAS_A.ALARMS.PROFILER_INIT_A AND NOT "DB2120_MPP_ITC_IPC".RESET_FAULTS AND NOT "DB7300_INTERLOCK_GENERAL".GENERAL_MACHINE.FROM_CELL_TO_MACHINE_GENERAL.MEAS_STA_RESET)) AND "DB7258_UNIT_3_STA_MEAS_A_ENABLE_DISABLE".ENABLED;
   "DB426_ALARMS_WARNINGS".UNIT_03.FACE_R_MEASURING."724244" := "DB16000_OPC_UA_TRIGGER_ALARM".CLIENT.U3_MEAS_STA_MEAS_A.ALARMS.PROFILER_INIT_A;
END_REGION

REGION Network 27: UNIT 3 MEASURING STATION FACE A RUN OUT ANALYSIS ALARM
   RUNG wire#powerrail
      { S7_Templates := "SrcType := Int" } EQ_Contact(in1 := "DB16006_U3_MEAS_STA_MEAS_A_CLIENT_INTERFACE".U03_FACE_A_MEAS_Read.Variable.Status, in2 := -1)
      Contact( "DB16006_U3_MEAS_STA_MEAS_A_CLIENT_INTERFACE".U03_FACE_A_MEAS_Read.Variable.RunOutAnalysis )
      wire#w1
      Contact( "DB7258_UNIT_3_STA_MEAS_A_ENABLE_DISABLE".ENABLED )
      wire#w2
      Coil( "DB16000_OPC_UA_TRIGGER_ALARM".CLIENT.U3_MEAS_STA_MEAS_A.ALARMS.RUNOUT_A )
   END_RUNG
   RUNG wire#powerrail
      Contact( "DB16000_OPC_UA_TRIGGER_ALARM".CLIENT.U3_MEAS_STA_MEAS_A.ALARMS.RUNOUT_A )
      I_Contact( "DB2120_MPP_ITC_IPC".RESET_FAULTS )
      I_Contact( "DB7300_INTERLOCK_GENERAL".GENERAL_MACHINE.FROM_CELL_TO_MACHINE_GENERAL.MEAS_STA_RESET )
   END_RUNG wire#w1
   RUNG wire#w2
      Coil( "DB426_ALARMS_WARNINGS".UNIT_03.FACE_R_MEASURING."724245" )
   END_RUNG
   // the same network as SCL:
   "DB16000_OPC_UA_TRIGGER_ALARM".CLIENT.U3_MEAS_STA_MEAS_A.ALARMS.RUNOUT_A := ((("DB16006_U3_MEAS_STA_MEAS_A_CLIENT_INTERFACE".U03_FACE_A_MEAS_Read.Variable.Status = (-1)) AND "DB16006_U3_MEAS_STA_MEAS_A_CLIENT_INTERFACE".U03_FACE_A_MEAS_Read.Variable.RunOutAnalysis) OR ("DB16000_OPC_UA_TRIGGER_ALARM".CLIENT.U3_MEAS_STA_MEAS_A.ALARMS.RUNOUT_A AND NOT "DB2120_MPP_ITC_IPC".RESET_FAULTS AND NOT "DB7300_INTERLOCK_GENERAL".GENERAL_MACHINE.FROM_CELL_TO_MACHINE_GENERAL.MEAS_STA_RESET)) AND "DB7258_UNIT_3_STA_MEAS_A_ENABLE_DISABLE".ENABLED;
   "DB426_ALARMS_WARNINGS".UNIT_03.FACE_R_MEASURING."724245" := "DB16000_OPC_UA_TRIGGER_ALARM".CLIENT.U3_MEAS_STA_MEAS_A.ALARMS.RUNOUT_A;
END_REGION

REGION Network 28: UNIT 3 MEASURING STATION FACE A UMBRELLA ANALYSIS ALARM
   RUNG wire#powerrail
      { S7_Templates := "SrcType := Int" } EQ_Contact(in1 := "DB16006_U3_MEAS_STA_MEAS_A_CLIENT_INTERFACE".U03_FACE_A_MEAS_Read.Variable.Status, in2 := -1)
      Contact( "DB16006_U3_MEAS_STA_MEAS_A_CLIENT_INTERFACE".U03_FACE_A_MEAS_Read.Variable.UmbrellaAnalysis )
      wire#w1
      Contact( "DB7258_UNIT_3_STA_MEAS_A_ENABLE_DISABLE".ENABLED )
      wire#w2
      Coil( "DB16000_OPC_UA_TRIGGER_ALARM".CLIENT.U3_MEAS_STA_MEAS_A.ALARMS.UMBRELLA_A )
   END_RUNG
   RUNG wire#powerrail
      Contact( "DB16000_OPC_UA_TRIGGER_ALARM".CLIENT.U3_MEAS_STA_MEAS_A.ALARMS.UMBRELLA_A )
      I_Contact( "DB2120_MPP_ITC_IPC".RESET_FAULTS )
      I_Contact( "DB7300_INTERLOCK_GENERAL".GENERAL_MACHINE.FROM_CELL_TO_MACHINE_GENERAL.MEAS_STA_RESET )
   END_RUNG wire#w1
   RUNG wire#w2
      Coil( "DB426_ALARMS_WARNINGS".UNIT_03.FACE_R_MEASURING."724246" )
   END_RUNG
   // the same network as SCL:
   "DB16000_OPC_UA_TRIGGER_ALARM".CLIENT.U3_MEAS_STA_MEAS_A.ALARMS.UMBRELLA_A := ((("DB16006_U3_MEAS_STA_MEAS_A_CLIENT_INTERFACE".U03_FACE_A_MEAS_Read.Variable.Status = (-1)) AND "DB16006_U3_MEAS_STA_MEAS_A_CLIENT_INTERFACE".U03_FACE_A_MEAS_Read.Variable.UmbrellaAnalysis) OR ("DB16000_OPC_UA_TRIGGER_ALARM".CLIENT.U3_MEAS_STA_MEAS_A.ALARMS.UMBRELLA_A AND NOT "DB2120_MPP_ITC_IPC".RESET_FAULTS AND NOT "DB7300_INTERLOCK_GENERAL".GENERAL_MACHINE.FROM_CELL_TO_MACHINE_GENERAL.MEAS_STA_RESET)) AND "DB7258_UNIT_3_STA_MEAS_A_ENABLE_DISABLE".ENABLED;
   "DB426_ALARMS_WARNINGS".UNIT_03.FACE_R_MEASURING."724246" := "DB16000_OPC_UA_TRIGGER_ALARM".CLIENT.U3_MEAS_STA_MEAS_A.ALARMS.UMBRELLA_A;
END_REGION

REGION Network 29: UNIT 3 MEASURING STATION FACE A LAYER GROWTH ANALYSIS ALARM
   RUNG wire#powerrail
      { S7_Templates := "SrcType := Int" } EQ_Contact(in1 := "DB16006_U3_MEAS_STA_MEAS_A_CLIENT_INTERFACE".U03_FACE_A_MEAS_Read.Variable.Status, in2 := -1)
      Contact( "M_ZERO" )
      wire#w1
      Contact( "DB7258_UNIT_3_STA_MEAS_A_ENABLE_DISABLE".ENABLED )
      wire#w2
      Coil( "DB16000_OPC_UA_TRIGGER_ALARM".CLIENT.U3_MEAS_STA_MEAS_A.ALARMS.LAYER_GROWTH_A )
   END_RUNG
   RUNG wire#powerrail
      Contact( "DB16000_OPC_UA_TRIGGER_ALARM".CLIENT.U3_MEAS_STA_MEAS_A.ALARMS.LAYER_GROWTH_A )
      I_Contact( "DB2120_MPP_ITC_IPC".RESET_FAULTS )
      I_Contact( "DB7300_INTERLOCK_GENERAL".GENERAL_MACHINE.FROM_CELL_TO_MACHINE_GENERAL.MEAS_STA_RESET )
   END_RUNG wire#w1
   RUNG wire#w2
      Coil( "DB426_ALARMS_WARNINGS".UNIT_03.FACE_R_MEASURING."724247" )
   END_RUNG
   // the same network as SCL:
   "DB16000_OPC_UA_TRIGGER_ALARM".CLIENT.U3_MEAS_STA_MEAS_A.ALARMS.LAYER_GROWTH_A := ((("DB16006_U3_MEAS_STA_MEAS_A_CLIENT_INTERFACE".U03_FACE_A_MEAS_Read.Variable.Status = (-1)) AND "M_ZERO") OR ("DB16000_OPC_UA_TRIGGER_ALARM".CLIENT.U3_MEAS_STA_MEAS_A.ALARMS.LAYER_GROWTH_A AND NOT "DB2120_MPP_ITC_IPC".RESET_FAULTS AND NOT "DB7300_INTERLOCK_GENERAL".GENERAL_MACHINE.FROM_CELL_TO_MACHINE_GENERAL.MEAS_STA_RESET)) AND "DB7258_UNIT_3_STA_MEAS_A_ENABLE_DISABLE".ENABLED;
   "DB426_ALARMS_WARNINGS".UNIT_03.FACE_R_MEASURING."724247" := "DB16000_OPC_UA_TRIGGER_ALARM".CLIENT.U3_MEAS_STA_MEAS_A.ALARMS.LAYER_GROWTH_A;
END_REGION

REGION Network 30: UNIT 3 MEASURING STATION FACE A SURFACE DEFECTS ANALYSIS ALARM
   RUNG wire#powerrail
      { S7_Templates := "SrcType := Int" } EQ_Contact(in1 := "DB16006_U3_MEAS_STA_MEAS_A_CLIENT_INTERFACE".U03_FACE_A_MEAS_Read.Variable.Status, in2 := -1)
      Contact( "DB16006_U3_MEAS_STA_MEAS_A_CLIENT_INTERFACE".U03_FACE_A_MEAS_Read.Variable.SurfaceDefectsAnalysis )
      wire#w1
      Contact( "DB7258_UNIT_3_STA_MEAS_A_ENABLE_DISABLE".ENABLED )
      wire#w2
      Coil( "DB16000_OPC_UA_TRIGGER_ALARM".CLIENT.U3_MEAS_STA_MEAS_A.ALARMS.SURFACE_DEFECTS_A )
   END_RUNG
   RUNG wire#powerrail
      Contact( "DB16000_OPC_UA_TRIGGER_ALARM".CLIENT.U3_MEAS_STA_MEAS_A.ALARMS.SURFACE_DEFECTS_A )
      I_Contact( "DB2120_MPP_ITC_IPC".RESET_FAULTS )
      I_Contact( "DB7300_INTERLOCK_GENERAL".GENERAL_MACHINE.FROM_CELL_TO_MACHINE_GENERAL.MEAS_STA_RESET )
   END_RUNG wire#w1
   RUNG wire#w2
      Coil( "DB426_ALARMS_WARNINGS".UNIT_03.FACE_R_MEASURING."724248" )
   END_RUNG
   // the same network as SCL:
   "DB16000_OPC_UA_TRIGGER_ALARM".CLIENT.U3_MEAS_STA_MEAS_A.ALARMS.SURFACE_DEFECTS_A := ((("DB16006_U3_MEAS_STA_MEAS_A_CLIENT_INTERFACE".U03_FACE_A_MEAS_Read.Variable.Status = (-1)) AND "DB16006_U3_MEAS_STA_MEAS_A_CLIENT_INTERFACE".U03_FACE_A_MEAS_Read.Variable.SurfaceDefectsAnalysis) OR ("DB16000_OPC_UA_TRIGGER_ALARM".CLIENT.U3_MEAS_STA_MEAS_A.ALARMS.SURFACE_DEFECTS_A AND NOT "DB2120_MPP_ITC_IPC".RESET_FAULTS AND NOT "DB7300_INTERLOCK_GENERAL".GENERAL_MACHINE.FROM_CELL_TO_MACHINE_GENERAL.MEAS_STA_RESET)) AND "DB7258_UNIT_3_STA_MEAS_A_ENABLE_DISABLE".ENABLED;
   "DB426_ALARMS_WARNINGS".UNIT_03.FACE_R_MEASURING."724248" := "DB16000_OPC_UA_TRIGGER_ALARM".CLIENT.U3_MEAS_STA_MEAS_A.ALARMS.SURFACE_DEFECTS_A;
END_REGION

REGION Network 31: UNIT 3 MEASURING STATION FACE A STORAGE ERROR ALARM
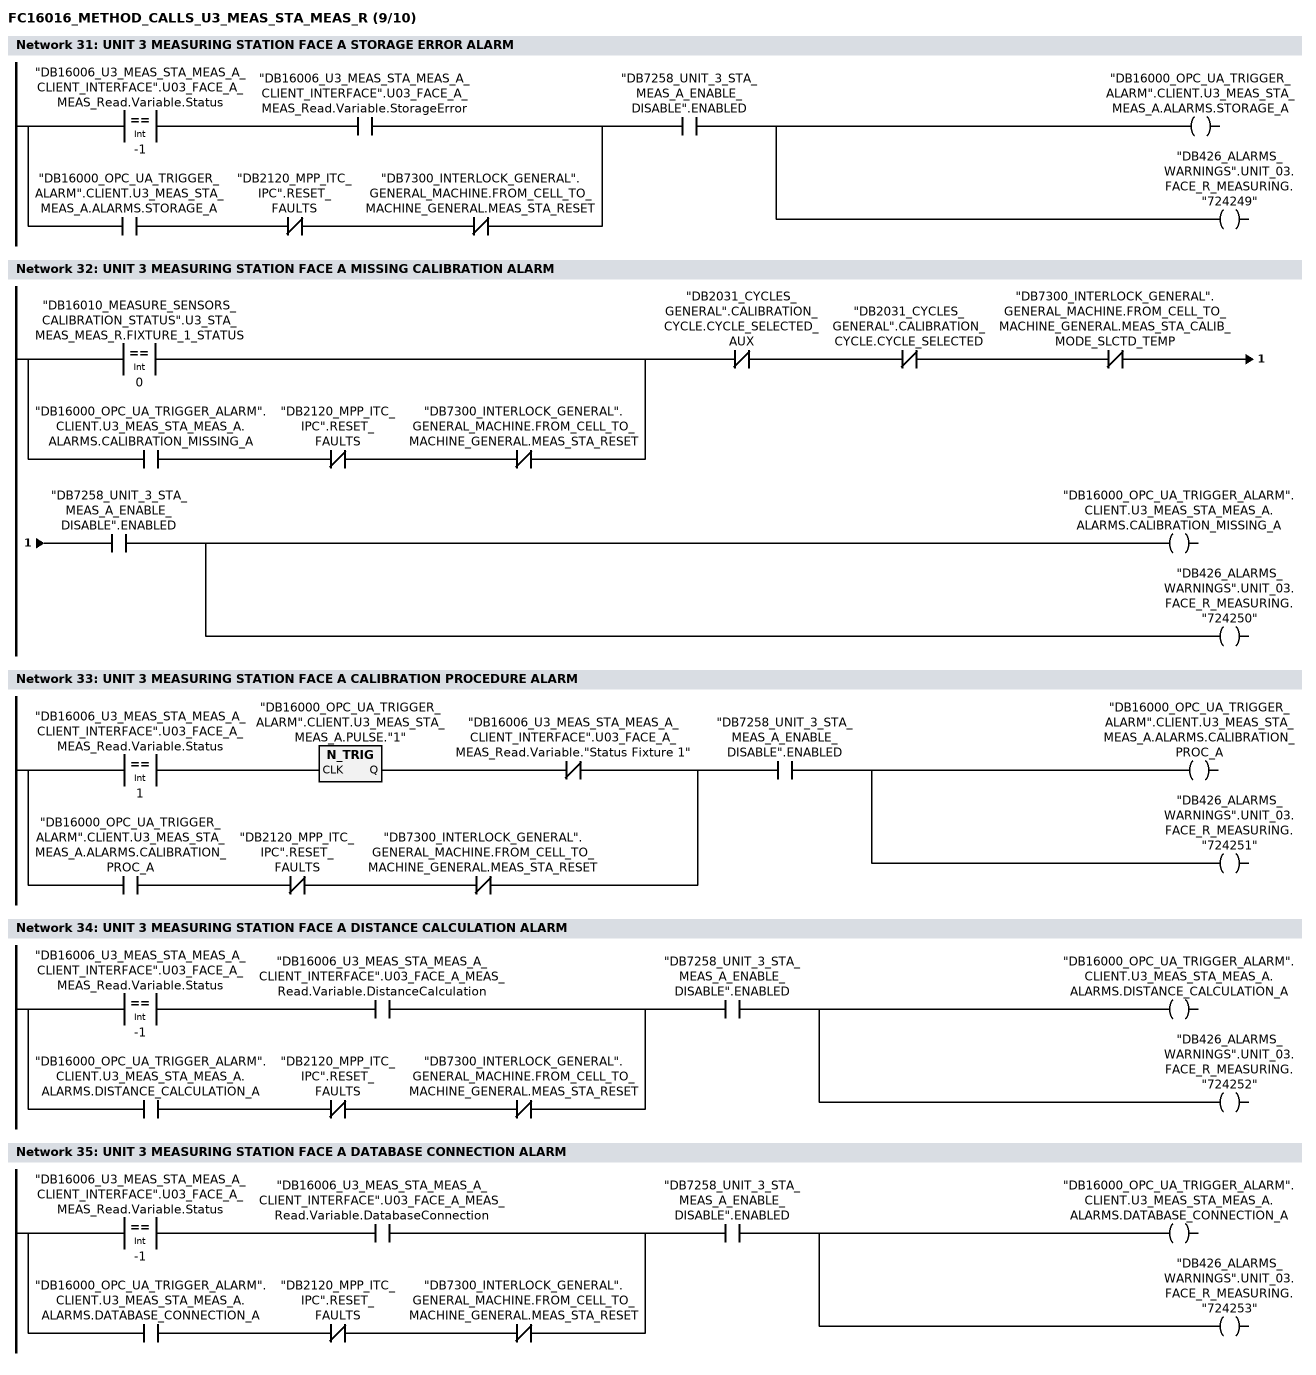
   RUNG wire#powerrail
      { S7_Templates := "SrcType := Int" } EQ_Contact(in1 := "DB16006_U3_MEAS_STA_MEAS_A_CLIENT_INTERFACE".U03_FACE_A_MEAS_Read.Variable.Status, in2 := -1)
      Contact( "DB16006_U3_MEAS_STA_MEAS_A_CLIENT_INTERFACE".U03_FACE_A_MEAS_Read.Variable.StorageError )
      wire#w1
      Contact( "DB7258_UNIT_3_STA_MEAS_A_ENABLE_DISABLE".ENABLED )
      wire#w2
      Coil( "DB16000_OPC_UA_TRIGGER_ALARM".CLIENT.U3_MEAS_STA_MEAS_A.ALARMS.STORAGE_A )
   END_RUNG
   RUNG wire#powerrail
      Contact( "DB16000_OPC_UA_TRIGGER_ALARM".CLIENT.U3_MEAS_STA_MEAS_A.ALARMS.STORAGE_A )
      I_Contact( "DB2120_MPP_ITC_IPC".RESET_FAULTS )
      I_Contact( "DB7300_INTERLOCK_GENERAL".GENERAL_MACHINE.FROM_CELL_TO_MACHINE_GENERAL.MEAS_STA_RESET )
   END_RUNG wire#w1
   RUNG wire#w2
      Coil( "DB426_ALARMS_WARNINGS".UNIT_03.FACE_R_MEASURING."724249" )
   END_RUNG
   // the same network as SCL:
   "DB16000_OPC_UA_TRIGGER_ALARM".CLIENT.U3_MEAS_STA_MEAS_A.ALARMS.STORAGE_A := ((("DB16006_U3_MEAS_STA_MEAS_A_CLIENT_INTERFACE".U03_FACE_A_MEAS_Read.Variable.Status = (-1)) AND "DB16006_U3_MEAS_STA_MEAS_A_CLIENT_INTERFACE".U03_FACE_A_MEAS_Read.Variable.StorageError) OR ("DB16000_OPC_UA_TRIGGER_ALARM".CLIENT.U3_MEAS_STA_MEAS_A.ALARMS.STORAGE_A AND NOT "DB2120_MPP_ITC_IPC".RESET_FAULTS AND NOT "DB7300_INTERLOCK_GENERAL".GENERAL_MACHINE.FROM_CELL_TO_MACHINE_GENERAL.MEAS_STA_RESET)) AND "DB7258_UNIT_3_STA_MEAS_A_ENABLE_DISABLE".ENABLED;
   "DB426_ALARMS_WARNINGS".UNIT_03.FACE_R_MEASURING."724249" := "DB16000_OPC_UA_TRIGGER_ALARM".CLIENT.U3_MEAS_STA_MEAS_A.ALARMS.STORAGE_A;
END_REGION

REGION Network 32: UNIT 3 MEASURING STATION FACE A MISSING CALIBRATION ALARM
   RUNG wire#powerrail
      { S7_Templates := "SrcType := Int" } EQ_Contact(in1 := "DB16010_MEASURE_SENSORS_CALIBRATION_STATUS".U3_STA_MEAS_MEAS_R.FIXTURE_1_STATUS, in2 := 0)
      wire#w1
      I_Contact( "DB2031_CYCLES_GENERAL".CALIBRATION_CYCLE.CYCLE_SELECTED_AUX )
      I_Contact( "DB2031_CYCLES_GENERAL".CALIBRATION_CYCLE.CYCLE_SELECTED )
      I_Contact( "DB7300_INTERLOCK_GENERAL".GENERAL_MACHINE.FROM_CELL_TO_MACHINE_GENERAL.MEAS_STA_CALIB_MODE_SLCTD_TEMP )
      Contact( "DB7258_UNIT_3_STA_MEAS_A_ENABLE_DISABLE".ENABLED )
      wire#w2
      Coil( "DB16000_OPC_UA_TRIGGER_ALARM".CLIENT.U3_MEAS_STA_MEAS_A.ALARMS.CALIBRATION_MISSING_A )
   END_RUNG
   RUNG wire#powerrail
      Contact( "DB16000_OPC_UA_TRIGGER_ALARM".CLIENT.U3_MEAS_STA_MEAS_A.ALARMS.CALIBRATION_MISSING_A )
      I_Contact( "DB2120_MPP_ITC_IPC".RESET_FAULTS )
      I_Contact( "DB7300_INTERLOCK_GENERAL".GENERAL_MACHINE.FROM_CELL_TO_MACHINE_GENERAL.MEAS_STA_RESET )
   END_RUNG wire#w1
   RUNG wire#w2
      Coil( "DB426_ALARMS_WARNINGS".UNIT_03.FACE_R_MEASURING."724250" )
   END_RUNG
   // the same network as SCL:
   "DB16000_OPC_UA_TRIGGER_ALARM".CLIENT.U3_MEAS_STA_MEAS_A.ALARMS.CALIBRATION_MISSING_A := (("DB16010_MEASURE_SENSORS_CALIBRATION_STATUS".U3_STA_MEAS_MEAS_R.FIXTURE_1_STATUS = 0) OR ("DB16000_OPC_UA_TRIGGER_ALARM".CLIENT.U3_MEAS_STA_MEAS_A.ALARMS.CALIBRATION_MISSING_A AND NOT "DB2120_MPP_ITC_IPC".RESET_FAULTS AND NOT "DB7300_INTERLOCK_GENERAL".GENERAL_MACHINE.FROM_CELL_TO_MACHINE_GENERAL.MEAS_STA_RESET)) AND NOT "DB2031_CYCLES_GENERAL".CALIBRATION_CYCLE.CYCLE_SELECTED_AUX AND NOT "DB2031_CYCLES_GENERAL".CALIBRATION_CYCLE.CYCLE_SELECTED AND NOT "DB7300_INTERLOCK_GENERAL".GENERAL_MACHINE.FROM_CELL_TO_MACHINE_GENERAL.MEAS_STA_CALIB_MODE_SLCTD_TEMP AND "DB7258_UNIT_3_STA_MEAS_A_ENABLE_DISABLE".ENABLED;
   "DB426_ALARMS_WARNINGS".UNIT_03.FACE_R_MEASURING."724250" := "DB16000_OPC_UA_TRIGGER_ALARM".CLIENT.U3_MEAS_STA_MEAS_A.ALARMS.CALIBRATION_MISSING_A;
END_REGION

REGION Network 33: UNIT 3 MEASURING STATION FACE A CALIBRATION PROCEDURE ALARM
   RUNG wire#powerrail
      { S7_Templates := "SrcType := Int" } EQ_Contact(in1 := "DB16006_U3_MEAS_STA_MEAS_A_CLIENT_INTERFACE".U03_FACE_A_MEAS_Read.Variable.Status, in2 := 1)
      N_Trig( "DB16000_OPC_UA_TRIGGER_ALARM".CLIENT.U3_MEAS_STA_MEAS_A.PULSE."1" )
      I_Contact( "DB16006_U3_MEAS_STA_MEAS_A_CLIENT_INTERFACE".U03_FACE_A_MEAS_Read.Variable."Status Fixture 1" )
      wire#w1
      Contact( "DB7258_UNIT_3_STA_MEAS_A_ENABLE_DISABLE".ENABLED )
      wire#w2
      Coil( "DB16000_OPC_UA_TRIGGER_ALARM".CLIENT.U3_MEAS_STA_MEAS_A.ALARMS.CALIBRATION_PROC_A )
   END_RUNG
   RUNG wire#powerrail
      Contact( "DB16000_OPC_UA_TRIGGER_ALARM".CLIENT.U3_MEAS_STA_MEAS_A.ALARMS.CALIBRATION_PROC_A )
      I_Contact( "DB2120_MPP_ITC_IPC".RESET_FAULTS )
      I_Contact( "DB7300_INTERLOCK_GENERAL".GENERAL_MACHINE.FROM_CELL_TO_MACHINE_GENERAL.MEAS_STA_RESET )
   END_RUNG wire#w1
   RUNG wire#w2
      Coil( "DB426_ALARMS_WARNINGS".UNIT_03.FACE_R_MEASURING."724251" )
   END_RUNG
   // the same network as SCL:
   #_w1 := "DB16006_U3_MEAS_STA_MEAS_A_CLIENT_INTERFACE".U03_FACE_A_MEAS_Read.Variable.Status = 1;
   #_w2 := NOT #_w1 AND "DB16000_OPC_UA_TRIGGER_ALARM".CLIENT.U3_MEAS_STA_MEAS_A.PULSE."1";   // falling edge
   "DB16000_OPC_UA_TRIGGER_ALARM".CLIENT.U3_MEAS_STA_MEAS_A.PULSE."1" := #_w1;
   "DB16000_OPC_UA_TRIGGER_ALARM".CLIENT.U3_MEAS_STA_MEAS_A.ALARMS.CALIBRATION_PROC_A := ((#_w2 AND NOT "DB16006_U3_MEAS_STA_MEAS_A_CLIENT_INTERFACE".U03_FACE_A_MEAS_Read.Variable."Status Fixture 1") OR ("DB16000_OPC_UA_TRIGGER_ALARM".CLIENT.U3_MEAS_STA_MEAS_A.ALARMS.CALIBRATION_PROC_A AND NOT "DB2120_MPP_ITC_IPC".RESET_FAULTS AND NOT "DB7300_INTERLOCK_GENERAL".GENERAL_MACHINE.FROM_CELL_TO_MACHINE_GENERAL.MEAS_STA_RESET)) AND "DB7258_UNIT_3_STA_MEAS_A_ENABLE_DISABLE".ENABLED;
   "DB426_ALARMS_WARNINGS".UNIT_03.FACE_R_MEASURING."724251" := "DB16000_OPC_UA_TRIGGER_ALARM".CLIENT.U3_MEAS_STA_MEAS_A.ALARMS.CALIBRATION_PROC_A;
END_REGION

REGION Network 34: UNIT 3 MEASURING STATION FACE A DISTANCE CALCULATION ALARM
   RUNG wire#powerrail
      { S7_Templates := "SrcType := Int" } EQ_Contact(in1 := "DB16006_U3_MEAS_STA_MEAS_A_CLIENT_INTERFACE".U03_FACE_A_MEAS_Read.Variable.Status, in2 := -1)
      Contact( "DB16006_U3_MEAS_STA_MEAS_A_CLIENT_INTERFACE".U03_FACE_A_MEAS_Read.Variable.DistanceCalculation )
      wire#w1
      Contact( "DB7258_UNIT_3_STA_MEAS_A_ENABLE_DISABLE".ENABLED )
      wire#w2
      Coil( "DB16000_OPC_UA_TRIGGER_ALARM".CLIENT.U3_MEAS_STA_MEAS_A.ALARMS.DISTANCE_CALCULATION_A )
   END_RUNG
   RUNG wire#powerrail
      Contact( "DB16000_OPC_UA_TRIGGER_ALARM".CLIENT.U3_MEAS_STA_MEAS_A.ALARMS.DISTANCE_CALCULATION_A )
      I_Contact( "DB2120_MPP_ITC_IPC".RESET_FAULTS )
      I_Contact( "DB7300_INTERLOCK_GENERAL".GENERAL_MACHINE.FROM_CELL_TO_MACHINE_GENERAL.MEAS_STA_RESET )
   END_RUNG wire#w1
   RUNG wire#w2
      Coil( "DB426_ALARMS_WARNINGS".UNIT_03.FACE_R_MEASURING."724252" )
   END_RUNG
   // the same network as SCL:
   "DB16000_OPC_UA_TRIGGER_ALARM".CLIENT.U3_MEAS_STA_MEAS_A.ALARMS.DISTANCE_CALCULATION_A := ((("DB16006_U3_MEAS_STA_MEAS_A_CLIENT_INTERFACE".U03_FACE_A_MEAS_Read.Variable.Status = (-1)) AND "DB16006_U3_MEAS_STA_MEAS_A_CLIENT_INTERFACE".U03_FACE_A_MEAS_Read.Variable.DistanceCalculation) OR ("DB16000_OPC_UA_TRIGGER_ALARM".CLIENT.U3_MEAS_STA_MEAS_A.ALARMS.DISTANCE_CALCULATION_A AND NOT "DB2120_MPP_ITC_IPC".RESET_FAULTS AND NOT "DB7300_INTERLOCK_GENERAL".GENERAL_MACHINE.FROM_CELL_TO_MACHINE_GENERAL.MEAS_STA_RESET)) AND "DB7258_UNIT_3_STA_MEAS_A_ENABLE_DISABLE".ENABLED;
   "DB426_ALARMS_WARNINGS".UNIT_03.FACE_R_MEASURING."724252" := "DB16000_OPC_UA_TRIGGER_ALARM".CLIENT.U3_MEAS_STA_MEAS_A.ALARMS.DISTANCE_CALCULATION_A;
END_REGION

REGION Network 35: UNIT 3 MEASURING STATION FACE A DATABASE CONNECTION ALARM
   RUNG wire#powerrail
      { S7_Templates := "SrcType := Int" } EQ_Contact(in1 := "DB16006_U3_MEAS_STA_MEAS_A_CLIENT_INTERFACE".U03_FACE_A_MEAS_Read.Variable.Status, in2 := -1)
      Contact( "DB16006_U3_MEAS_STA_MEAS_A_CLIENT_INTERFACE".U03_FACE_A_MEAS_Read.Variable.DatabaseConnection )
      wire#w1
      Contact( "DB7258_UNIT_3_STA_MEAS_A_ENABLE_DISABLE".ENABLED )
      wire#w2
      Coil( "DB16000_OPC_UA_TRIGGER_ALARM".CLIENT.U3_MEAS_STA_MEAS_A.ALARMS.DATABASE_CONNECTION_A )
   END_RUNG
   RUNG wire#powerrail
      Contact( "DB16000_OPC_UA_TRIGGER_ALARM".CLIENT.U3_MEAS_STA_MEAS_A.ALARMS.DATABASE_CONNECTION_A )
      I_Contact( "DB2120_MPP_ITC_IPC".RESET_FAULTS )
      I_Contact( "DB7300_INTERLOCK_GENERAL".GENERAL_MACHINE.FROM_CELL_TO_MACHINE_GENERAL.MEAS_STA_RESET )
   END_RUNG wire#w1
   RUNG wire#w2
      Coil( "DB426_ALARMS_WARNINGS".UNIT_03.FACE_R_MEASURING."724253" )
   END_RUNG
   // the same network as SCL:
   "DB16000_OPC_UA_TRIGGER_ALARM".CLIENT.U3_MEAS_STA_MEAS_A.ALARMS.DATABASE_CONNECTION_A := ((("DB16006_U3_MEAS_STA_MEAS_A_CLIENT_INTERFACE".U03_FACE_A_MEAS_Read.Variable.Status = (-1)) AND "DB16006_U3_MEAS_STA_MEAS_A_CLIENT_INTERFACE".U03_FACE_A_MEAS_Read.Variable.DatabaseConnection) OR ("DB16000_OPC_UA_TRIGGER_ALARM".CLIENT.U3_MEAS_STA_MEAS_A.ALARMS.DATABASE_CONNECTION_A AND NOT "DB2120_MPP_ITC_IPC".RESET_FAULTS AND NOT "DB7300_INTERLOCK_GENERAL".GENERAL_MACHINE.FROM_CELL_TO_MACHINE_GENERAL.MEAS_STA_RESET)) AND "DB7258_UNIT_3_STA_MEAS_A_ENABLE_DISABLE".ENABLED;
   "DB426_ALARMS_WARNINGS".UNIT_03.FACE_R_MEASURING."724253" := "DB16000_OPC_UA_TRIGGER_ALARM".CLIENT.U3_MEAS_STA_MEAS_A.ALARMS.DATABASE_CONNECTION_A;
END_REGION

REGION Network 36: UNIT 3 MEASURING PLC PC MINOR VERSIONS MISMATCH WARNING
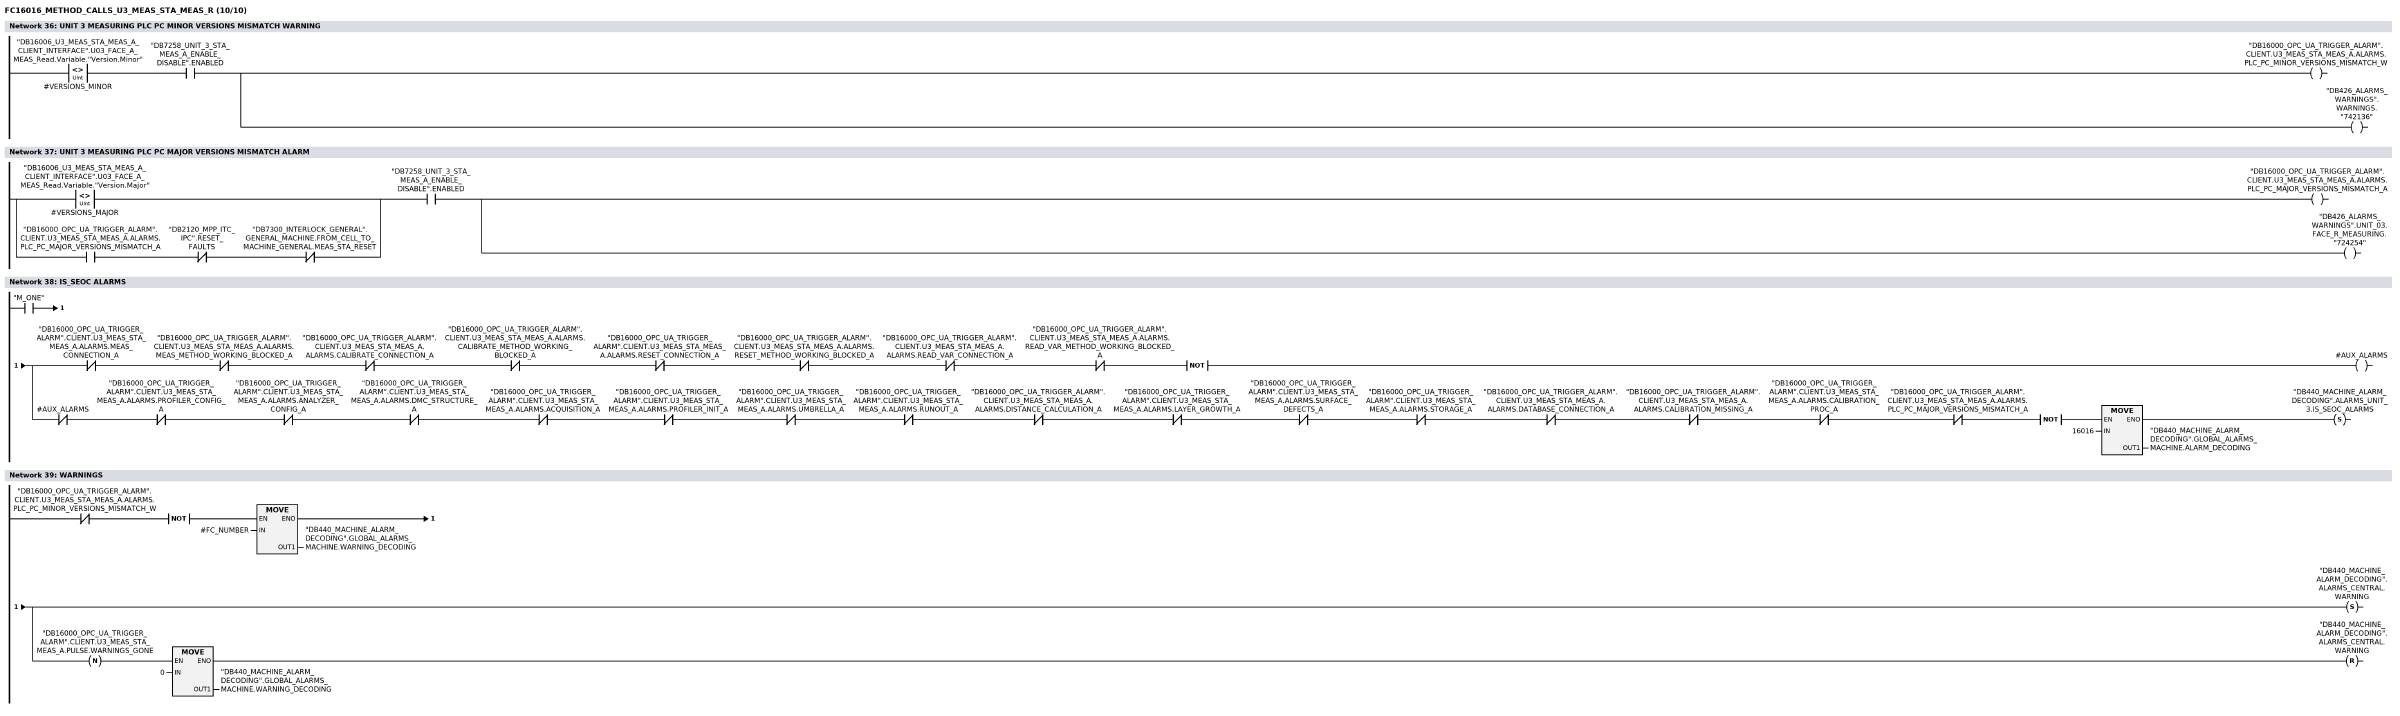
   RUNG wire#powerrail
      { S7_Templates := "SrcType := UInt" } NE_Contact(in1 := "DB16006_U3_MEAS_STA_MEAS_A_CLIENT_INTERFACE".U03_FACE_A_MEAS_Read.Variable."Version.Minor", in2 := #VERSIONS_MINOR)
      Contact( "DB7258_UNIT_3_STA_MEAS_A_ENABLE_DISABLE".ENABLED )
      wire#w1
      Coil( "DB16000_OPC_UA_TRIGGER_ALARM".CLIENT.U3_MEAS_STA_MEAS_A.ALARMS.PLC_PC_MINOR_VERSIONS_MISMATCH_W )
   END_RUNG
   RUNG wire#w1
      Coil( "DB426_ALARMS_WARNINGS".WARNINGS."742136" )
   END_RUNG
   // the same network as SCL:
   "DB16000_OPC_UA_TRIGGER_ALARM".CLIENT.U3_MEAS_STA_MEAS_A.ALARMS.PLC_PC_MINOR_VERSIONS_MISMATCH_W := ("DB16006_U3_MEAS_STA_MEAS_A_CLIENT_INTERFACE".U03_FACE_A_MEAS_Read.Variable."Version.Minor" <> #VERSIONS_MINOR) AND "DB7258_UNIT_3_STA_MEAS_A_ENABLE_DISABLE".ENABLED;
   "DB426_ALARMS_WARNINGS".WARNINGS."742136" := "DB16000_OPC_UA_TRIGGER_ALARM".CLIENT.U3_MEAS_STA_MEAS_A.ALARMS.PLC_PC_MINOR_VERSIONS_MISMATCH_W;
END_REGION

REGION Network 37: UNIT 3 MEASURING PLC PC MAJOR VERSIONS MISMATCH ALARM
   RUNG wire#powerrail
      { S7_Templates := "SrcType := UInt" } NE_Contact(in1 := "DB16006_U3_MEAS_STA_MEAS_A_CLIENT_INTERFACE".U03_FACE_A_MEAS_Read.Variable."Version.Major", in2 := #VERSIONS_MAJOR)
      wire#w1
      Contact( "DB7258_UNIT_3_STA_MEAS_A_ENABLE_DISABLE".ENABLED )
      wire#w2
      Coil( "DB16000_OPC_UA_TRIGGER_ALARM".CLIENT.U3_MEAS_STA_MEAS_A.ALARMS.PLC_PC_MAJOR_VERSIONS_MISMATCH_A )
   END_RUNG
   RUNG wire#powerrail
      Contact( "DB16000_OPC_UA_TRIGGER_ALARM".CLIENT.U3_MEAS_STA_MEAS_A.ALARMS.PLC_PC_MAJOR_VERSIONS_MISMATCH_A )
      I_Contact( "DB2120_MPP_ITC_IPC".RESET_FAULTS )
      I_Contact( "DB7300_INTERLOCK_GENERAL".GENERAL_MACHINE.FROM_CELL_TO_MACHINE_GENERAL.MEAS_STA_RESET )
   END_RUNG wire#w1
   RUNG wire#w2
      Coil( "DB426_ALARMS_WARNINGS".UNIT_03.FACE_R_MEASURING."724254" )
   END_RUNG
   // the same network as SCL:
   "DB16000_OPC_UA_TRIGGER_ALARM".CLIENT.U3_MEAS_STA_MEAS_A.ALARMS.PLC_PC_MAJOR_VERSIONS_MISMATCH_A := (("DB16006_U3_MEAS_STA_MEAS_A_CLIENT_INTERFACE".U03_FACE_A_MEAS_Read.Variable."Version.Major" <> #VERSIONS_MAJOR) OR ("DB16000_OPC_UA_TRIGGER_ALARM".CLIENT.U3_MEAS_STA_MEAS_A.ALARMS.PLC_PC_MAJOR_VERSIONS_MISMATCH_A AND NOT "DB2120_MPP_ITC_IPC".RESET_FAULTS AND NOT "DB7300_INTERLOCK_GENERAL".GENERAL_MACHINE.FROM_CELL_TO_MACHINE_GENERAL.MEAS_STA_RESET)) AND "DB7258_UNIT_3_STA_MEAS_A_ENABLE_DISABLE".ENABLED;
   "DB426_ALARMS_WARNINGS".UNIT_03.FACE_R_MEASURING."724254" := "DB16000_OPC_UA_TRIGGER_ALARM".CLIENT.U3_MEAS_STA_MEAS_A.ALARMS.PLC_PC_MAJOR_VERSIONS_MISMATCH_A;
END_REGION

REGION Network 38: IS_SEOC ALARMS
   RUNG wire#powerrail
      Contact( "M_ONE" )
      wire#w1
      I_Contact( "DB16000_OPC_UA_TRIGGER_ALARM".CLIENT.U3_MEAS_STA_MEAS_A.ALARMS.MEAS_CONNECTION_A )
      I_Contact( "DB16000_OPC_UA_TRIGGER_ALARM".CLIENT.U3_MEAS_STA_MEAS_A.ALARMS.MEAS_METHOD_WORKING_BLOCKED_A )
      I_Contact( "DB16000_OPC_UA_TRIGGER_ALARM".CLIENT.U3_MEAS_STA_MEAS_A.ALARMS.CALIBRATE_CONNECTION_A )
      I_Contact( "DB16000_OPC_UA_TRIGGER_ALARM".CLIENT.U3_MEAS_STA_MEAS_A.ALARMS.CALIBRATE_METHOD_WORKING_BLOCKED_A )
      I_Contact( "DB16000_OPC_UA_TRIGGER_ALARM".CLIENT.U3_MEAS_STA_MEAS_A.ALARMS.RESET_CONNECTION_A )
      I_Contact( "DB16000_OPC_UA_TRIGGER_ALARM".CLIENT.U3_MEAS_STA_MEAS_A.ALARMS.RESET_METHOD_WORKING_BLOCKED_A )
      I_Contact( "DB16000_OPC_UA_TRIGGER_ALARM".CLIENT.U3_MEAS_STA_MEAS_A.ALARMS.READ_VAR_CONNECTION_A )
      I_Contact( "DB16000_OPC_UA_TRIGGER_ALARM".CLIENT.U3_MEAS_STA_MEAS_A.ALARMS.READ_VAR_METHOD_WORKING_BLOCKED_A )
      Not()
      Coil( #AUX_ALARMS )
   END_RUNG
   RUNG wire#w1
      I_Contact( #AUX_ALARMS )
      I_Contact( "DB16000_OPC_UA_TRIGGER_ALARM".CLIENT.U3_MEAS_STA_MEAS_A.ALARMS.PROFILER_CONFIG_A )
      I_Contact( "DB16000_OPC_UA_TRIGGER_ALARM".CLIENT.U3_MEAS_STA_MEAS_A.ALARMS.ANALYZER_CONFIG_A )
      I_Contact( "DB16000_OPC_UA_TRIGGER_ALARM".CLIENT.U3_MEAS_STA_MEAS_A.ALARMS.DMC_STRUCTURE_A )
      I_Contact( "DB16000_OPC_UA_TRIGGER_ALARM".CLIENT.U3_MEAS_STA_MEAS_A.ALARMS.ACQUISITION_A )
      I_Contact( "DB16000_OPC_UA_TRIGGER_ALARM".CLIENT.U3_MEAS_STA_MEAS_A.ALARMS.PROFILER_INIT_A )
      I_Contact( "DB16000_OPC_UA_TRIGGER_ALARM".CLIENT.U3_MEAS_STA_MEAS_A.ALARMS.UMBRELLA_A )
      I_Contact( "DB16000_OPC_UA_TRIGGER_ALARM".CLIENT.U3_MEAS_STA_MEAS_A.ALARMS.RUNOUT_A )
      I_Contact( "DB16000_OPC_UA_TRIGGER_ALARM".CLIENT.U3_MEAS_STA_MEAS_A.ALARMS.DISTANCE_CALCULATION_A )
      I_Contact( "DB16000_OPC_UA_TRIGGER_ALARM".CLIENT.U3_MEAS_STA_MEAS_A.ALARMS.LAYER_GROWTH_A )
      I_Contact( "DB16000_OPC_UA_TRIGGER_ALARM".CLIENT.U3_MEAS_STA_MEAS_A.ALARMS.SURFACE_DEFECTS_A )
      I_Contact( "DB16000_OPC_UA_TRIGGER_ALARM".CLIENT.U3_MEAS_STA_MEAS_A.ALARMS.STORAGE_A )
      I_Contact( "DB16000_OPC_UA_TRIGGER_ALARM".CLIENT.U3_MEAS_STA_MEAS_A.ALARMS.DATABASE_CONNECTION_A )
      I_Contact( "DB16000_OPC_UA_TRIGGER_ALARM".CLIENT.U3_MEAS_STA_MEAS_A.ALARMS.CALIBRATION_MISSING_A )
      I_Contact( "DB16000_OPC_UA_TRIGGER_ALARM".CLIENT.U3_MEAS_STA_MEAS_A.ALARMS.CALIBRATION_PROC_A )
      I_Contact( "DB16000_OPC_UA_TRIGGER_ALARM".CLIENT.U3_MEAS_STA_MEAS_A.ALARMS.PLC_PC_MAJOR_VERSIONS_MISMATCH_A )
      Not()
      Move(in := 16016, out1 => "DB440_MACHINE_ALARM_DECODING".GLOBAL_ALARMS_MACHINE.ALARM_DECODING)
      S_Coil( "DB440_MACHINE_ALARM_DECODING".ALARMS_UNIT_3.IS_SEOC_ALARMS )
   END_RUNG
   // the same network as SCL:
   #AUX_ALARMS := NOT ("M_ONE" AND NOT "DB16000_OPC_UA_TRIGGER_ALARM".CLIENT.U3_MEAS_STA_MEAS_A.ALARMS.MEAS_CONNECTION_A AND NOT "DB16000_OPC_UA_TRIGGER_ALARM".CLIENT.U3_MEAS_STA_MEAS_A.ALARMS.MEAS_METHOD_WORKING_BLOCKED_A AND NOT "DB16000_OPC_UA_TRIGGER_ALARM".CLIENT.U3_MEAS_STA_MEAS_A.ALARMS.CALIBRATE_CONNECTION_A AND NOT "DB16000_OPC_UA_TRIGGER_ALARM".CLIENT.U3_MEAS_STA_MEAS_A.ALARMS.CALIBRATE_METHOD_WORKING_BLOCKED_A AND NOT "DB16000_OPC_UA_TRIGGER_ALARM".CLIENT.U3_MEAS_STA_MEAS_A.ALARMS.RESET_CONNECTION_A AND NOT "DB16000_OPC_UA_TRIGGER_ALARM".CLIENT.U3_MEAS_STA_MEAS_A.ALARMS.RESET_METHOD_WORKING_BLOCKED_A AND NOT "DB16000_OPC_UA_TRIGGER_ALARM".CLIENT.U3_MEAS_STA_MEAS_A.ALARMS.READ_VAR_CONNECTION_A AND NOT "DB16000_OPC_UA_TRIGGER_ALARM".CLIENT.U3_MEAS_STA_MEAS_A.ALARMS.READ_VAR_METHOD_WORKING_BLOCKED_A);
   IF NOT ("M_ONE" AND NOT #AUX_ALARMS AND NOT "DB16000_OPC_UA_TRIGGER_ALARM".CLIENT.U3_MEAS_STA_MEAS_A.ALARMS.PROFILER_CONFIG_A AND NOT "DB16000_OPC_UA_TRIGGER_ALARM".CLIENT.U3_MEAS_STA_MEAS_A.ALARMS.ANALYZER_CONFIG_A AND NOT "DB16000_OPC_UA_TRIGGER_ALARM".CLIENT.U3_MEAS_STA_MEAS_A.ALARMS.DMC_STRUCTURE_A AND NOT "DB16000_OPC_UA_TRIGGER_ALARM".CLIENT.U3_MEAS_STA_MEAS_A.ALARMS.ACQUISITION_A AND NOT "DB16000_OPC_UA_TRIGGER_ALARM".CLIENT.U3_MEAS_STA_MEAS_A.ALARMS.PROFILER_INIT_A AND NOT "DB16000_OPC_UA_TRIGGER_ALARM".CLIENT.U3_MEAS_STA_MEAS_A.ALARMS.UMBRELLA_A AND NOT "DB16000_OPC_UA_TRIGGER_ALARM".CLIENT.U3_MEAS_STA_MEAS_A.ALARMS.RUNOUT_A AND NOT "DB16000_OPC_UA_TRIGGER_ALARM".CLIENT.U3_MEAS_STA_MEAS_A.ALARMS.DISTANCE_CALCULATION_A AND NOT "DB16000_OPC_UA_TRIGGER_ALARM".CLIENT.U3_MEAS_STA_MEAS_A.ALARMS.LAYER_GROWTH_A AND NOT "DB16000_OPC_UA_TRIGGER_ALARM".CLIENT.U3_MEAS_STA_MEAS_A.ALARMS.SURFACE_DEFECTS_A AND NOT "DB16000_OPC_UA_TRIGGER_ALARM".CLIENT.U3_MEAS_STA_MEAS_A.ALARMS.STORAGE_A AND NOT "DB16000_OPC_UA_TRIGGER_ALARM".CLIENT.U3_MEAS_STA_MEAS_A.ALARMS.DATABASE_CONNECTION_A AND NOT "DB16000_OPC_UA_TRIGGER_ALARM".CLIENT.U3_MEAS_STA_MEAS_A.ALARMS.CALIBRATION_MISSING_A AND NOT "DB16000_OPC_UA_TRIGGER_ALARM".CLIENT.U3_MEAS_STA_MEAS_A.ALARMS.CALIBRATION_PROC_A AND NOT "DB16000_OPC_UA_TRIGGER_ALARM".CLIENT.U3_MEAS_STA_MEAS_A.ALARMS.PLC_PC_MAJOR_VERSIONS_MISMATCH_A) THEN
       "DB440_MACHINE_ALARM_DECODING".GLOBAL_ALARMS_MACHINE.ALARM_DECODING := 16016;
       "DB440_MACHINE_ALARM_DECODING".ALARMS_UNIT_3.IS_SEOC_ALARMS := TRUE;
   END_IF;
END_REGION

REGION Network 39: WARNINGS
   RUNG wire#powerrail
      I_Contact( "DB16000_OPC_UA_TRIGGER_ALARM".CLIENT.U3_MEAS_STA_MEAS_A.ALARMS.PLC_PC_MINOR_VERSIONS_MISMATCH_W )
      Not()
      Move(in := #FC_NUMBER, out1 => "DB440_MACHINE_ALARM_DECODING".GLOBAL_ALARMS_MACHINE.WARNING_DECODING)
      wire#w1
      S_Coil( "DB440_MACHINE_ALARM_DECODING".ALARMS_CENTRAL.WARNING )
   END_RUNG
   RUNG wire#w1
      N_Trig( "DB16000_OPC_UA_TRIGGER_ALARM".CLIENT.U3_MEAS_STA_MEAS_A.PULSE.WARNINGS_GONE )
      Move(in := 0, out1 => "DB440_MACHINE_ALARM_DECODING".GLOBAL_ALARMS_MACHINE.WARNING_DECODING)
      R_Coil( "DB440_MACHINE_ALARM_DECODING".ALARMS_CENTRAL.WARNING )
   END_RUNG
   // the same network as SCL:
   #_w1 := NOT (NOT "DB16000_OPC_UA_TRIGGER_ALARM".CLIENT.U3_MEAS_STA_MEAS_A.ALARMS.PLC_PC_MINOR_VERSIONS_MISMATCH_W);
   IF #_w1 THEN
       "DB440_MACHINE_ALARM_DECODING".GLOBAL_ALARMS_MACHINE.WARNING_DECODING := #FC_NUMBER;
       "DB440_MACHINE_ALARM_DECODING".ALARMS_CENTRAL.WARNING := TRUE;
   END_IF;
   #_w2 := NOT #_w1 AND "DB16000_OPC_UA_TRIGGER_ALARM".CLIENT.U3_MEAS_STA_MEAS_A.PULSE.WARNINGS_GONE;   // falling edge
   "DB16000_OPC_UA_TRIGGER_ALARM".CLIENT.U3_MEAS_STA_MEAS_A.PULSE.WARNINGS_GONE := #_w1;
   IF #_w2 THEN
       "DB440_MACHINE_ALARM_DECODING".GLOBAL_ALARMS_MACHINE.WARNING_DECODING := 0;
       "DB440_MACHINE_ALARM_DECODING".ALARMS_CENTRAL.WARNING := FALSE;
   END_IF;
END_REGION
END_FUNCTION
